KUKA KRL program: EPS_2_251806_MH04A_A_20260213065133.src

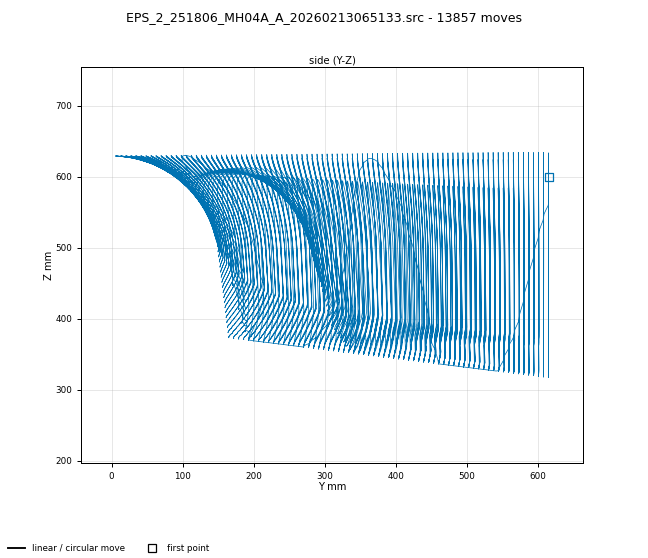
[picture p0: tool path of EPS_2_251806_MH04A_A_20260213065133.src, 13857 of 13859 moves have a stored position in this frame; points joined in program order, loops and branches not executed]
&ACCESS RVP
&REL 4
&COMMENT QRS 19112012
&PARAM EDITMASK = *
DEF PART()
EXT BAS (BAS_COMMAND :IN,REAL :IN )
INT I
BAS (#INITMOV,0 )

;KUKA QRS Post kuka4.cps  Date:22-06-2017 !

File_ID=3013

QRS_PRE_INIT()

;Init var - Until changes are made in qrs_pre_init
Outlet_Square_prg=0
Inlet_1_Square_prg=0
Inlet_2_Square_prg=0
Inlet_3_Square_prg=0
Inlet_4_Square_prg=0
Inlet_5_Square_prg=0

Outlet_1={X 0.000, Y 527.380, Z 509.000, B 0.000, E1 0.000 }
Inlet_1={X 0.000, Y 533.670, Z 484.000, B 0.000, E1 90.000 }
Inlet_2={X 0.000, Y 528.100, Z 499.000, B 0.000, E1 180.000 }
Outlet_1_type=251
Inlet_1_type=201
Inlet_2_type=251
;QRS#1=Sidecore dimensions
;QRS#2=250-10" PVC SDR 35
;QRS#3=200-8" PVC SDR 35
;QRS#4=250-10" PVC SDR 35
;QRS#5=
;QRS#6=
;QRS#7=
;QRS#8=
;QRS#9=14M PSX
;QRS#10=12-08 PSX
;QRS#11=14M PSX
;QRS#12=
;QRS#13=
;QRS#14=
;QRS#15=
;QRS#16=1220x127x914 3'
;QRS#17=EPS Height
;QRS#18=634,5
;QRS#19=*
;QRS#20= UPDATED VERSION 22-06-2017
;QRS#21=*
Outlet_Square=0100
Inlet_1_Square=0100
Inlet_2_Square=0100
Inlet_3_Square=0
Inlet_4_Square=0
Inlet_5_Square=0
Mill_Square=1
Outlet_Square_Prg=205
Inlet_1_Square_prg=204
Inlet_2_Square_prg=205

QRS_INIT()

$ADVANCE=5

; T1
PTP {E1 173.497,E2 173.497}
PTP {X 0,Y 615.499,A -85,B 0,C 180,E1 173.497,E2 173.497,E3 0,E4 0,E5 0,E6 0}
QRS_SPEED_INIT()
LIN {X 0,Y 615.499,Z 600,A -85,B 0,C 180,E1 173.497,E2 173.497,E3 0,E4 0,E5 0,E6 0} C_VEL
LIN {X 0,Y 615.499,Z 575.226,A -85,B 0,C 180,E1 173.497,E2 173.497} C_VEL
LIN {X 0,Y 615.499,Z 564.346,A -85,B 0,C 180,E1 173.497,E2 173.497} C_VEL
LIN {X 0,Y 615.497,Z 562.701,A -85,B 0,C 180,E1 173.417,E2 173.417} C_VEL
LIN {X 0,Y 615.497,Z 555.036,A -85,B 0,C 180,E1 172.455,E2 172.455} C_VEL
LIN {X 0,Y 615.498,Z 545.258,A -85,B 0,C 180,E1 171.463,E2 171.463} C_VEL
LIN {X 0,Y 615.497,Z 534.992,A -85,B 0,C 180,E1 170.636,E2 170.636} C_VEL
LIN {X 0,Y 615.479,Z 523.431,A -85,B 0,C 180,E1 169.888,E2 169.888} C_VEL
LIN {X 0,Y 615.498,Z 511.575,A -85,B 0,C 180,E1 169.293,E2 169.293} C_VEL
LIN {X 0,Y 615.483,Z 498.658,A -85,B 0,C 180,E1 168.807,E2 168.807} C_VEL
LIN {X 0,Y 615.49,Z 486.055,A -85,B 0,C 180,E1 168.473,E2 168.473} C_VEL
LIN {X 0,Y 615.489,Z 472.927,A -85,B 0,C 180,E1 168.264,E2 168.264} C_VEL
LIN {X 0,Y 615.486,Z 372.646,A -85,B 0,C 180,E1 167.072,E2 167.072} C_VEL
LIN {X 0,Y 615.491,Z 353.313,A -85,B 0,C 180,E1 164.265,E2 164.265} C_VEL
LIN {X 0,Y 615.488,Z 333.804,A -85,B 0,C 180,E1 161.396,E2 161.396} C_VEL
LIN {X 0,Y 615.479,Z 317.312,A -85,B 0,C 180,E1 158.919,E2 158.919} C_VEL
LIN {X 0,Y 615.487,Z 317.309,A -85,B 0,C 180,E1 156.444,E2 156.444} C_VEL
LIN {X 0,Y 615.483,Z 317.322,A -85,B 0,C 180,E1 153.556,E2 153.556} C_VEL
LIN {X 0,Y 615.471,Z 317.317,A -85,B 0,C 180,E1 151.341,E2 151.341} C_VEL
LIN {X 0,Y 615.479,Z 317.31,A -85,B 0,C 180,E1 148.916,E2 148.916} C_VEL
LIN {X 0,Y 615.496,Z 317.326,A -85,B 0,C 180,E1 145.978,E2 145.978} C_VEL
LIN {X 0,Y 615.464,Z 317.319,A -85,B 0,C 180,E1 143.573,E2 143.573} C_VEL
LIN {X 0,Y 615.474,Z 317.312,A -85,B 0,C 180,E1 140.94,E2 140.94} C_VEL
LIN {X 0,Y 615.471,Z 317.322,A -85,B 0,C 180,E1 137.922,E2 137.922} C_VEL
LIN {X 0,Y 615.46,Z 317.321,A -85,B 0,C 180,E1 135.848,E2 135.848} C_VEL
LIN {X 0,Y 615.467,Z 317.314,A -85,B 0,C 180,E1 133.045,E2 133.045} C_VEL
LIN {X 0,Y 615.461,Z 317.323,A -85,B 0,C 180,E1 130.086,E2 130.086} C_VEL
LIN {X 0,Y 615.449,Z 317.322,A -85,B 0,C 180,E1 128.007,E2 128.007} C_VEL
LIN {X 0,Y 615.432,Z 317.321,A -85,B 0,C 180,E1 125.62,E2 125.62} C_VEL
LIN {X 0,Y 615.447,Z 317.32,A -85,B 0,C 180,E1 123.239,E2 123.239} C_VEL
LIN {X 0,Y 615.486,Z 317.32,A -85,B 0,C 180,E1 120.921,E2 120.921} C_VEL
LIN {X 0,Y 615.457,Z 317.325,A -85,B 0,C 180,E1 118.445,E2 118.445} C_VEL
LIN {X 0,Y 615.45,Z 317.325,A -85,B 0,C 180,E1 116.447,E2 116.447} C_VEL
LIN {X 0,Y 615.412,Z 317.325,A -85,B 0,C 180,E1 113.992,E2 113.992} C_VEL
LIN {X 0,Y 615.422,Z 317.46,A -85,B 0,C 180,E1 111.633,E2 111.633} C_VEL
LIN {X 0,Y 615.493,Z 336.679,A -85,B 0,C 180,E1 108.992,E2 108.992} C_VEL
LIN {X 0,Y 615.483,Z 357.59,A -85,B 0,C 180,E1 106.166,E2 106.166} C_VEL
LIN {X 0,Y 615.491,Z 362.222,A -85,B 0,C 180,E1 105.545,E2 105.545} C_VEL
LIN {X 0,Y 615.497,Z 499.149,A -85,B 0,C 180,E1 103.905,E2 103.905} C_VEL
LIN {X 0,Y 615.493,Z 512.715,A -85,B 0,C 180,E1 103.622,E2 103.622} C_VEL
LIN {X 0,Y 615.495,Z 526.464,A -85,B 0,C 180,E1 103.202,E2 103.202} C_VEL
LIN {X 0,Y 615.495,Z 538.882,A -85,B 0,C 180,E1 102.698,E2 102.698} C_VEL
LIN {X 0,Y 615.495,Z 551.827,A -85,B 0,C 180,E1 102.029,E2 102.029} C_VEL
LIN {X 0,Y 615.499,Z 563.546,A -85,B 0,C 180,E1 101.277,E2 101.277} C_VEL
LIN {X 0,Y 615.498,Z 575.215,A -85,B 0,C 180,E1 100.361,E2 100.361} C_VEL
LIN {X 0,Y 615.497,Z 585.641,A -85,B 0,C 180,E1 99.365,E2 99.365} C_VEL
LIN {X 0,Y 615.496,Z 594.232,A -85,B 0,C 180,E1 98.372,E2 98.372} C_VEL
LIN {X 0,Y 615.495,Z 602.447,A -85,B 0,C 180,E1 97.216,E2 97.216} C_VEL
LIN {X 0,Y 615.496,Z 608.178,A -85,B 0,C 180,E1 96.228,E2 96.228} C_VEL
LIN {X 0,Y 615.491,Z 612.884,A -85,B 0,C 180,E1 95.242,E2 95.242} C_VEL
LIN {X 0,Y 615.496,Z 617.754,A -85,B 0,C 180,E1 93.929,E2 93.929} C_VEL
LIN {X 0,Y 615.496,Z 621.152,A -85,B 0,C 180,E1 92.619,E2 92.619} C_VEL
LIN {X 0,Y 615.493,Z 623.173,A -85,B 0,C 180,E1 91.31,E2 91.31} C_VEL
LIN {X 0,Y 615.494,Z 623.884,A -85,B 0,C 180,E1 90.001,E2 90.001} C_VEL
LIN {X 0,Y 615.49,Z 623.281,A -85,B 0,C 180,E1 88.692,E2 88.692} C_VEL
LIN {X 0,Y 615.493,Z 621.353,A -85,B 0,C 180,E1 87.383,E2 87.383} C_VEL
LIN {X 0,Y 615.496,Z 618.049,A -85,B 0,C 180,E1 86.073,E2 86.073} C_VEL
LIN {X 0,Y 615.496,Z 613.278,A -85,B 0,C 180,E1 84.76,E2 84.76} C_VEL
LIN {X 0,Y 615.494,Z 606.88,A -85,B 0,C 180,E1 83.444,E2 83.444} C_VEL
LIN {X 0,Y 615.496,Z 599.751,A -85,B 0,C 180,E1 82.291,E2 82.291} C_VEL
LIN {X 0,Y 615.497,Z 592.28,A -85,B 0,C 180,E1 81.299,E2 81.299} C_VEL
LIN {X 0,Y 615.495,Z 583.302,A -85,B 0,C 180,E1 80.305,E2 80.305} C_VEL
LIN {X 0,Y 615.499,Z 572.212,A -85,B 0,C 180,E1 79.291,E2 79.291} C_VEL
LIN {X 0,Y 615.498,Z 561.297,A -85,B 0,C 180,E1 78.475,E2 78.475} C_VEL
LIN {X 0,Y 615.488,Z 549.004,A -85,B 0,C 180,E1 77.722,E2 77.722} C_VEL
LIN {X 0,Y 615.498,Z 537.171,A -85,B 0,C 180,E1 77.136,E2 77.136} C_VEL
LIN {X 0,Y 615.492,Z 524.254,A -85,B 0,C 180,E1 76.632,E2 76.632} C_VEL
LIN {X 0,Y 615.495,Z 511.288,A -85,B 0,C 180,E1 76.253,E2 76.253} C_VEL
LIN {X 0,Y 615.493,Z 497.999,A -85,B 0,C 180,E1 75.988,E2 75.988} C_VEL
LIN {X 0,Y 615.493,Z 362.117,A -85,B 0,C 180,E1 74.351,E2 74.351} C_VEL
LIN {X 0,Y 615.477,Z 341.407,A -85,B 0,C 180,E1 71.559,E2 71.559} C_VEL
LIN {X 0,Y 615.491,Z 322.099,A -85,B 0,C 180,E1 68.921,E2 68.921} C_VEL
LIN {X 0,Y 615.426,Z 317.323,A -85,B 0,C 180,E1 68.237,E2 68.237} C_VEL
LIN {X 0,Y 615.432,Z 317.321,A -85,B 0,C 180,E1 65.727,E2 65.727} C_VEL
LIN {X 0,Y 615.473,Z 317.325,A -85,B 0,C 180,E1 62.824,E2 62.824} C_VEL
LIN {X 0,Y 615.42,Z 317.323,A -85,B 0,C 180,E1 60.217,E2 60.217} C_VEL
LIN {X 0,Y 615.425,Z 317.323,A -85,B 0,C 180,E1 58.313,E2 58.313} C_VEL
LIN {X 0,Y 615.422,Z 317.322,A -85,B 0,C 180,E1 55.976,E2 55.976} C_VEL
LIN {X 0,Y 615.449,Z 317.321,A -85,B 0,C 180,E1 53.574,E2 53.574} C_VEL
LIN {X 0,Y 615.478,Z 317.325,A -85,B 0,C 180,E1 50.939,E2 50.939} C_VEL
LIN {X 0,Y 615.432,Z 317.323,A -85,B 0,C 180,E1 48.523,E2 48.523} C_VEL
LIN {X 0,Y 615.422,Z 317.322,A -85,B 0,C 180,E1 46.009,E2 46.009} C_VEL
LIN {X 0,Y 615.499,Z 317.321,A -85,B 0,C 180,E1 43.244,E2 43.244} C_VEL
LIN {X 0,Y 615.433,Z 317.324,A -85,B 0,C 180,E1 40.611,E2 40.611} C_VEL
LIN {X 0,Y 615.462,Z 317.324,A -85,B 0,C 180,E1 38.906,E2 38.906} C_VEL
LIN {X 0,Y 615.422,Z 317.323,A -85,B 0,C 180,E1 36.429,E2 36.429} C_VEL
LIN {X 0,Y 615.467,Z 317.321,A -85,B 0,C 180,E1 33.534,E2 33.534} C_VEL
LIN {X 0,Y 615.456,Z 317.324,A -85,B 0,C 180,E1 30.922,E2 30.922} C_VEL
LIN {X 0,Y 615.419,Z 317.323,A -85,B 0,C 180,E1 28.442,E2 28.442} C_VEL
LIN {X 0,Y 615.419,Z 317.323,A -85,B 0,C 180,E1 26.447,E2 26.447} C_VEL
LIN {X 0,Y 615.426,Z 317.323,A -85,B 0,C 180,E1 23.999,E2 23.999} C_VEL
LIN {X 0,Y 615.489,Z 317.322,A -85,B 0,C 180,E1 21.432,E2 21.432} C_VEL
LIN {X 0,Y 615.421,Z 317.324,A -85,B 0,C 180,E1 18.591,E2 18.591} C_VEL
LIN {X 0,Y 615.415,Z 317.324,A -85,B 0,C 180,E1 16.414,E2 16.414} C_VEL
LIN {X 0,Y 615.435,Z 317.323,A -85,B 0,C 180,E1 13.92,E2 13.92} C_VEL
LIN {X 0,Y 615.433,Z 317.325,A -85,B 0,C 180,E1 10.87,E2 10.87} C_VEL
LIN {X 0,Y 615.416,Z 317.324,A -85,B 0,C 180,E1 8.538,E2 8.538} C_VEL
LIN {X 0,Y 615.413,Z 317.324,A -85,B 0,C 180,E1 6.533,E2 6.533} C_VEL
LIN {X 0,Y 615.415,Z 317.324,A -85,B 0,C 180,E1 4.585,E2 4.585} C_VEL
LIN {X 0,Y 615.417,Z 317.324,A -85,B 0,C 180,E1 2.618,E2 2.618} C_VEL
LIN {X 0,Y 615.417,Z 317.324,A -85,B 0,C 180,E1 0.654,E2 0.654} C_VEL
LIN {X 0,Y 615.418,Z 317.324,A -85,B 0,C 180,E1 -1.309,E2 -1.309} C_VEL
LIN {X 0,Y 615.419,Z 317.324,A -85,B 0,C 180,E1 -3.273,E2 -3.273} C_VEL
LIN {X 0,Y 615.419,Z 317.324,A -85,B 0,C 180,E1 -5.242,E2 -5.242} C_VEL
LIN {X 0,Y 615.417,Z 317.325,A -85,B 0,C 180,E1 -7.216,E2 -7.216} C_VEL
LIN {X 0,Y 615.419,Z 317.325,A -85,B 0,C 180,E1 -9.2,E2 -9.2} C_VEL
LIN {X 0,Y 615.419,Z 317.324,A -85,B 0,C 180,E1 -11.194,E2 -11.194} C_VEL
LIN {X 0,Y 615.418,Z 317.324,A -85,B 0,C 180,E1 -13.203,E2 -13.203} C_VEL
LIN {X 0,Y 615.416,Z 317.324,A -85,B 0,C 180,E1 -15.228,E2 -15.228} C_VEL
LIN {X 0,Y 615.414,Z 317.324,A -85,B 0,C 180,E1 -17.273,E2 -17.273} C_VEL
LIN {X 0,Y 615.412,Z 317.324,A -85,B 0,C 180,E1 -19.34,E2 -19.34} C_VEL
LIN {X 0,Y 615.411,Z 317.324,A -85,B 0,C 180,E1 -21.435,E2 -21.435} C_VEL
LIN {X 0,Y 615.411,Z 317.325,A -85,B 0,C 180,E1 -23.559,E2 -23.559} C_VEL
LIN {X 0,Y 615.489,Z 317.325,A -85,B 0,C 180,E1 -26.444,E2 -26.444} C_VEL
LIN {X 0,Y 615.455,Z 317.325,A -85,B 0,C 180,E1 -28.66,E2 -28.66} C_VEL
LIN {X 0,Y 615.416,Z 317.325,A -85,B 0,C 180,E1 -31.078,E2 -31.078} C_VEL
LIN {X 0,Y 615.41,Z 317.325,A -85,B 0,C 180,E1 -33.241,E2 -33.241} C_VEL
LIN {X 0,Y 615.435,Z 317.325,A -85,B 0,C 180,E1 -35.83,E2 -35.83} C_VEL
LIN {X 0,Y 615.465,Z 317.325,A -85,B 0,C 180,E1 -38.07,E2 -38.07} C_VEL
LIN {X 0,Y 615.45,Z 317.325,A -85,B 0,C 180,E1 -40.609,E2 -40.609} C_VEL
LIN {X 0,Y 615.413,Z 317.325,A -85,B 0,C 180,E1 -43.042,E2 -43.042} C_VEL
LIN {X 0,Y 615.411,Z 317.325,A -85,B 0,C 180,E1 -45.076,E2 -45.076} C_VEL
LIN {X 0,Y 615.424,Z 317.325,A -85,B 0,C 180,E1 -47.644,E2 -47.644} C_VEL
LIN {X 0,Y 615.488,Z 317.326,A -85,B 0,C 180,E1 -50.252,E2 -50.252} C_VEL
LIN {X 0,Y 615.427,Z 317.325,A -85,B 0,C 180,E1 -52.755,E2 -52.755} C_VEL
LIN {X 0,Y 615.41,Z 317.325,A -85,B 0,C 180,E1 -55.182,E2 -55.182} C_VEL
LIN {X 0,Y 615.433,Z 317.325,A -85,B 0,C 180,E1 -57.678,E2 -57.678} C_VEL
LIN {X 0,Y 615.439,Z 317.324,A -85,B 0,C 180,E1 -60.593,E2 -60.593} C_VEL
LIN {X 0,Y 615.413,Z 317.324,A -85,B 0,C 180,E1 -62.969,E2 -62.969} C_VEL
LIN {X 0,Y 615.412,Z 317.324,A -85,B 0,C 180,E1 -65.006,E2 -65.006} C_VEL
LIN {X 0,Y 615.418,Z 317.458,A -85,B 0,C 180,E1 -67.378,E2 -67.378} C_VEL
LIN {X 0,Y 615.484,Z 337.246,A -85,B 0,C 180,E1 -69.968,E2 -69.968} C_VEL
LIN {X 0,Y 615.486,Z 358.699,A -85,B 0,C 180,E1 -72.731,E2 -72.731} C_VEL
LIN {X 0,Y 615.493,Z 372.139,A -85,B 0,C 180,E1 -74.415,E2 -74.415} C_VEL
LIN {X 0,Y 615.499,Z 509.922,A -85,B 0,C 180,E1 -76.064,E2 -76.064} C_VEL
LIN {X 0,Y 615.495,Z 524.419,A -85,B 0,C 180,E1 -76.38,E2 -76.38} C_VEL
LIN {X 0,Y 615.489,Z 537.719,A -85,B 0,C 180,E1 -76.8,E2 -76.8} C_VEL
LIN {X 0,Y 615.498,Z 551.606,A -85,B 0,C 180,E1 -77.387,E2 -77.387} C_VEL
LIN {X 0,Y 615.495,Z 564.026,A -85,B 0,C 180,E1 -78.057,E2 -78.057} C_VEL
LIN {X 0,Y 615.499,Z 575.356,A -85,B 0,C 180,E1 -78.808,E2 -78.808} C_VEL
LIN {X 0,Y 615.498,Z 585.761,A -85,B 0,C 180,E1 -79.641,E2 -79.641} C_VEL
LIN {X 0,Y 615.496,Z 596.099,A -85,B 0,C 180,E1 -80.637,E2 -80.637} C_VEL
LIN {X 0,Y 615.497,Z 604.611,A -85,B 0,C 180,E1 -81.63,E2 -81.63} C_VEL
LIN {X 0,Y 615.496,Z 612.733,A -85,B 0,C 180,E1 -82.786,E2 -82.786} C_VEL
LIN {X 0,Y 615.496,Z 618.436,A -85,B 0,C 180,E1 -83.774,E2 -83.774} C_VEL
LIN {X 0,Y 615.495,Z 623.085,A -85,B 0,C 180,E1 -84.76,E2 -84.76} C_VEL
LIN {X 0,Y 615.494,Z 627.905,A -85,B 0,C 180,E1 -86.073,E2 -86.073} C_VEL
LIN {X 0,Y 615.496,Z 631.254,A -85,B 0,C 180,E1 -87.383,E2 -87.383} C_VEL
LIN {X 0,Y 615.489,Z 633.23,A -85,B 0,C 180,E1 -88.692,E2 -88.692} C_VEL
LIN {X 0,Y 615.493,Z 633.889,A -85,B 0,C 180,E1 -90.001,E2 -90.001} C_VEL
LIN {X 0,Y 615.489,Z 633.227,A -85,B 0,C 180,E1 -91.31,E2 -91.31} C_VEL
LIN {X 0,Y 615.496,Z 631.25,A -85,B 0,C 180,E1 -92.619,E2 -92.619} C_VEL
LIN {X 0,Y 615.494,Z 627.898,A -85,B 0,C 180,E1 -93.929,E2 -93.929} C_VEL
LIN {X 0,Y 615.495,Z 623.076,A -85,B 0,C 180,E1 -95.242,E2 -95.242} C_VEL
LIN {X 0,Y 615.496,Z 616.623,A -85,B 0,C 180,E1 -96.557,E2 -96.557} C_VEL
LIN {X 0,Y 615.497,Z 609.434,A -85,B 0,C 180,E1 -97.711,E2 -97.711} C_VEL
LIN {X 0,Y 615.497,Z 601.896,A -85,B 0,C 180,E1 -98.703,E2 -98.703} C_VEL
LIN {X 0,Y 615.495,Z 592.844,A -85,B 0,C 180,E1 -99.697,E2 -99.697} C_VEL
LIN {X 0,Y 615.497,Z 582.75,A -85,B 0,C 180,E1 -100.619,E2 -100.619} C_VEL
LIN {X 0,Y 615.498,Z 571.844,A -85,B 0,C 180,E1 -101.444,E2 -101.444} C_VEL
LIN {X 0,Y 615.489,Z 559.689,A -85,B 0,C 180,E1 -102.196,E2 -102.196} C_VEL
LIN {X 0,Y 615.498,Z 546.069,A -85,B 0,C 180,E1 -102.866,E2 -102.866} C_VEL
LIN {X 0,Y 615.49,Z 532.807,A -85,B 0,C 180,E1 -103.37,E2 -103.37} C_VEL
LIN {X 0,Y 615.494,Z 519.247,A -85,B 0,C 180,E1 -103.749,E2 -103.749} C_VEL
LIN {X 0,Y 615.496,Z 504.72,A -85,B 0,C 180,E1 -104.013,E2 -104.013} C_VEL
LIN {X 0,Y 615.494,Z 371.744,A -85,B 0,C 180,E1 -105.608,E2 -105.608} C_VEL
LIN {X 0,Y 615.482,Z 349.549,A -85,B 0,C 180,E1 -108.442,E2 -108.442} C_VEL
LIN {X 0,Y 615.485,Z 329.177,A -85,B 0,C 180,E1 -111.082,E2 -111.082} C_VEL
LIN {X 0,Y 615.419,Z 317.325,A -85,B 0,C 180,E1 -112.656,E2 -112.656} C_VEL
LIN {X 0,Y 615.423,Z 317.324,A -85,B 0,C 180,E1 -114.995,E2 -114.995} C_VEL
LIN {X 0,Y 615.443,Z 317.324,A -85,B 0,C 180,E1 -117.18,E2 -117.18} C_VEL
LIN {X 0,Y 615.457,Z 317.318,A -85,B 0,C 180,E1 -120.162,E2 -120.162} C_VEL
LIN {X 0,Y 615.446,Z 317.318,A -85,B 0,C 180,E1 -122.461,E2 -122.461} C_VEL
LIN {X 0,Y 615.456,Z 317.321,A -85,B 0,C 180,E1 -124.818,E2 -124.818} C_VEL
LIN {X 0,Y 615.492,Z 317.325,A -85,B 0,C 180,E1 -127.243,E2 -127.243} C_VEL
LIN {X 0,Y 615.473,Z 317.312,A -85,B 0,C 180,E1 -130.087,E2 -130.087} C_VEL
LIN {X 0,Y 615.468,Z 317.316,A -85,B 0,C 180,E1 -132.355,E2 -132.355} C_VEL
LIN {X 0,Y 615.486,Z 317.32,A -85,B 0,C 180,E1 -135.069,E2 -135.069} C_VEL
LIN {X 0,Y 615.487,Z 317.31,A -85,B 0,C 180,E1 -137.921,E2 -137.921} C_VEL
LIN {X 0,Y 615.484,Z 317.318,A -85,B 0,C 180,E1 -140.25,E2 -140.25} C_VEL
LIN {X 0,Y 615.464,Z 317.317,A -85,B 0,C 180,E1 -143.067,E2 -143.067} C_VEL
LIN {X 0,Y 615.467,Z 317.313,A -85,B 0,C 180,E1 -145.303,E2 -145.303} C_VEL
LIN {X 0,Y 615.494,Z 317.311,A -85,B 0,C 180,E1 -147.669,E2 -147.669} C_VEL
LIN {X 0,Y 615.454,Z 317.321,A -85,B 0,C 180,E1 -150.592,E2 -150.592} C_VEL
LIN {X 0,Y 615.441,Z 317.319,A -85,B 0,C 180,E1 -152.964,E2 -152.964} C_VEL
LIN {X 0,Y 615.495,Z 317.321,A -85,B 0,C 180,E1 -155.728,E2 -155.728} C_VEL
LIN {X 0,Y 615.479,Z 317.326,A -85,B 0,C 180,E1 -157.863,E2 -157.863} C_VEL
LIN {X 0,Y 615.433,Z 317.48,A -85,B 0,C 180,E1 -159.049,E2 -159.049} C_VEL
LIN {X 0,Y 615.496,Z 335.382,A -85,B 0,C 180,E1 -161.72,E2 -161.72} C_VEL
LIN {X 0,Y 615.498,Z 355.023,A -85,B 0,C 180,E1 -164.605,E2 -164.605} C_VEL
LIN {X 0,Y 615.49,Z 372.749,A -85,B 0,C 180,E1 -167.177,E2 -167.177} C_VEL
LIN {X 0,Y 615.493,Z 480.144,A -85,B 0,C 180,E1 -168.453,E2 -168.453} C_VEL
LIN {X 0,Y 615.491,Z 492.724,A -85,B 0,C 180,E1 -168.724,E2 -168.724} C_VEL
LIN {X 0,Y 615.491,Z 506.106,A -85,B 0,C 180,E1 -169.158,E2 -169.158} C_VEL
LIN {X 0,Y 615.492,Z 517.066,A -85,B 0,C 180,E1 -169.639,E2 -169.639} C_VEL
LIN {X 0,Y 615.482,Z 528.806,A -85,B 0,C 180,E1 -170.304,E2 -170.304} C_VEL
LIN {X 0,Y 615.499,Z 539.268,A -85,B 0,C 180,E1 -171.05,E2 -171.05} C_VEL
LIN {X 0,Y 615.498,Z 547.831,A -85,B 0,C 180,E1 -171.794,E2 -171.794} C_VEL
LIN {X 0,Y 615.498,Z 555.709,A -85,B 0,C 180,E1 -172.62,E2 -172.62} C_VEL
LIN {X 0,Y 615.497,Z 563.399,A -85,B 0,C 180,E1 -173.608,E2 -173.608} C_VEL
LIN {X 0,Y 615.498,Z 570.458,A -85,B 0,C 180,E1 -174.759,E2 -174.759} C_VEL
LIN {X 0,Y 615.493,Z 575.158,A -85,B 0,C 180,E1 -175.744,E2 -175.744} C_VEL
LIN {X 0,Y 615.496,Z 578.754,A -85,B 0,C 180,E1 -176.727,E2 -176.727} C_VEL
LIN {X 0,Y 615.496,Z 580.615,A -85,B 0,C 180,E1 -177.382,E2 -177.382} C_VEL
LIN {X 0,Y 615.497,Z 582.034,A -85,B 0,C 180,E1 -178.037,E2 -178.037} C_VEL
LIN {X 0,Y 615.496,Z 583.642,A -85,B 0,C 180,E1 -179.346,E2 -179.346} C_VEL
LIN {X 0,Y 615.494,Z 583.884,A -85,B 0,C 180,E1 -180,E2 -180} C_VEL
LIN {X 0,Y 615.496,Z 583.705,A -85,B 0,C 180,E1 -180.654,E2 -180.654} C_VEL
LIN {X 0,Y 615.496,Z 582.183,A -85,B 0,C 180,E1 -181.963,E2 -181.963} C_VEL
LIN {X 0,Y 615.498,Z 580.841,A -85,B 0,C 180,E1 -182.618,E2 -182.618} C_VEL
LIN {X 0,Y 615.497,Z 577.994,A -85,B 0,C 180,E1 -183.601,E2 -183.601} C_VEL
LIN {X 0,Y 615.499,Z 574.134,A -85,B 0,C 180,E1 -184.585,E2 -184.585} C_VEL
LIN {X 0,Y 615.498,Z 569.151,A -85,B 0,C 180,E1 -185.57,E2 -185.57} C_VEL
LIN {X 0,Y 615.497,Z 562.701,A -85,B 0,C 180,E1 -186.583,E2 -186.583} C_VEL
LIN {X 0,Y 614.829,Z 559.52,A -85,B 0,C 180,E1 -187.032,E2 -187.032} C_VEL
LIN {X 0,Y 611.988,Z 553.946,A -85,B 0,C 180,E1 -187.749,E2 -187.749} C_VEL
LIN {X 0,Y 609.138,Z 547.67,A -85,B 0,C 180,E1 -188.43,E2 -188.43} C_VEL
LIN {X 0,Y 608.477,Z 543.429,A -85,B 0,C 180,E1 -188.82,E2 -188.82} C_VEL
LIN {X 0,Y 608.489,Z 532.886,A -85,B 0,C 180,E1 -189.641,E2 -189.641} C_VEL
LIN {X 0,Y 608.49,Z 522.11,A -85,B 0,C 180,E1 -190.313,E2 -190.313} C_VEL
LIN {X 0,Y 608.52,Z 509.659,A -85,B 0,C 180,E1 -190.919,E2 -190.919} C_VEL
LIN {X 0,Y 608.522,Z 497.464,A -85,B 0,C 180,E1 -191.365,E2 -191.365} C_VEL
LIN {X 0,Y 608.549,Z 485.156,A -85,B 0,C 180,E1 -191.681,E2 -191.681} C_VEL
LIN {X 0,Y 608.556,Z 471.245,A -85,B 0,C 180,E1 -191.892,E2 -191.892} C_VEL
LIN {X 0,Y 608.466,Z 372.952,A -85,B 0,C 180,E1 -193.059,E2 -193.059} C_VEL
LIN {X 0,Y 608.492,Z 353.399,A -85,B 0,C 180,E1 -195.921,E2 -195.921} C_VEL
LIN {X 0,Y 608.515,Z 334.494,A -85,B 0,C 180,E1 -198.727,E2 -198.727} C_VEL
LIN {X 0,Y 608.476,Z 318.312,A -85,B 0,C 180,E1 -201.18,E2 -201.18} C_VEL
LIN {X 0,Y 608.465,Z 318.314,A -85,B 0,C 180,E1 -203.845,E2 -203.845} C_VEL
LIN {X 0,Y 608.443,Z 318.321,A -85,B 0,C 180,E1 -206.036,E2 -206.036} C_VEL
LIN {X 0,Y 608.464,Z 318.315,A -85,B 0,C 180,E1 -208.618,E2 -208.618} C_VEL
LIN {X 0,Y 608.449,Z 318.314,A -85,B 0,C 180,E1 -211.318,E2 -211.318} C_VEL
LIN {X 0,Y 608.477,Z 318.315,A -85,B 0,C 180,E1 -213.735,E2 -213.735} C_VEL
LIN {X 0,Y 608.447,Z 318.322,A -85,B 0,C 180,E1 -216.092,E2 -216.092} C_VEL
LIN {X 0,Y 608.427,Z 318.317,A -85,B 0,C 180,E1 -218.591,E2 -218.591} C_VEL
LIN {X 0,Y 608.462,Z 318.314,A -85,B 0,C 180,E1 -221.341,E2 -221.341} C_VEL
LIN {X 0,Y 608.462,Z 318.32,A -85,B 0,C 180,E1 -223.87,E2 -223.87} C_VEL
LIN {X 0,Y 608.445,Z 318.314,A -85,B 0,C 180,E1 -226.694,E2 -226.694} C_VEL
LIN {X 0,Y 608.427,Z 318.316,A -85,B 0,C 180,E1 -228.82,E2 -228.82} C_VEL
LIN {X 0,Y 608.445,Z 318.32,A -85,B 0,C 180,E1 -231.763,E2 -231.763} C_VEL
LIN {X 0,Y 608.434,Z 318.318,A -85,B 0,C 180,E1 -233.957,E2 -233.957} C_VEL
LIN {X 0,Y 608.415,Z 318.317,A -85,B 0,C 180,E1 -236.325,E2 -236.325} C_VEL
LIN {X 0,Y 608.438,Z 318.316,A -85,B 0,C 180,E1 -238.734,E2 -238.734} C_VEL
LIN {X 0,Y 608.41,Z 318.321,A -85,B 0,C 180,E1 -241.73,E2 -241.73} C_VEL
LIN {X 0,Y 608.394,Z 318.32,A -85,B 0,C 180,E1 -244.295,E2 -244.295} C_VEL
LIN {X 0,Y 608.421,Z 318.323,A -85,B 0,C 180,E1 -246.874,E2 -246.874} C_VEL
LIN {X 0,Y 608.402,Z 318.419,A -85,B 0,C 180,E1 -248.238,E2 -248.238} C_VEL
LIN {X 0,Y 608.546,Z 332.889,A -85,B 0,C 180,E1 -250.256,E2 -250.256} C_VEL
LIN {X 0,Y 608.505,Z 353.244,A -85,B 0,C 180,E1 -253.044,E2 -253.044} C_VEL
LIN {X 0,Y 608.512,Z 362.308,A -85,B 0,C 180,E1 -254.272,E2 -254.272} C_VEL
LIN {X 0,Y 608.614,Z 474.489,A -85,B 0,C 180,E1 -255.624,E2 -255.624} C_VEL
LIN {X 0,Y 608.611,Z 500.869,A -85,B 0,C 180,E1 -255.965,E2 -255.965} C_VEL
LIN {X 0,Y 608.6,Z 515.036,A -85,B 0,C 180,E1 -256.284,E2 -256.284} C_VEL
LIN {X 0,Y 608.576,Z 528.741,A -85,B 0,C 180,E1 -256.73,E2 -256.73} C_VEL
LIN {X 0,Y 608.545,Z 540.673,A -85,B 0,C 180,E1 -257.239,E2 -257.239} C_VEL
LIN {X 0,Y 608.534,Z 553.325,A -85,B 0,C 180,E1 -257.916,E2 -257.916} C_VEL
LIN {X 0,Y 608.5,Z 564.841,A -85,B 0,C 180,E1 -258.676,E2 -258.676} C_VEL
LIN {X 0,Y 608.495,Z 575.404,A -85,B 0,C 180,E1 -259.518,E2 -259.518} C_VEL
LIN {X 0,Y 608.48,Z 585.89,A -85,B 0,C 180,E1 -260.526,E2 -260.526} C_VEL
LIN {X 0,Y 608.463,Z 594.542,A -85,B 0,C 180,E1 -261.53,E2 -261.53} C_VEL
LIN {X 0,Y 608.461,Z 602.833,A -85,B 0,C 180,E1 -262.7,E2 -262.7} C_VEL
LIN {X 0,Y 608.443,Z 609.322,A -85,B 0,C 180,E1 -263.831,E2 -263.831} C_VEL
LIN {X 0,Y 608.437,Z 614.784,A -85,B 0,C 180,E1 -265.029,E2 -265.029} C_VEL
LIN {X 0,Y 608.434,Z 618.295,A -85,B 0,C 180,E1 -266.025,E2 -266.025} C_VEL
LIN {X 0,Y 608.424,Z 621.731,A -85,B 0,C 180,E1 -267.351,E2 -267.351} C_VEL
LIN {X 0,Y 608.446,Z 623.775,A -85,B 0,C 180,E1 -268.675,E2 -268.675} C_VEL
LIN {X 0,Y 608.434,Z 624.495,A -85,B 0,C 180,E1 -269.999,E2 -269.999} C_VEL
LIN {X 0,Y 608.443,Z 623.883,A -85,B 0,C 180,E1 -271.323,E2 -271.323} C_VEL
LIN {X 0,Y 608.421,Z 621.93,A -85,B 0,C 180,E1 -272.647,E2 -272.647} C_VEL
LIN {X 0,Y 608.434,Z 618.589,A -85,B 0,C 180,E1 -273.973,E2 -273.973} C_VEL
LIN {X 0,Y 608.44,Z 613.765,A -85,B 0,C 180,E1 -275.301,E2 -275.301} C_VEL
LIN {X 0,Y 608.438,Z 607.302,A -85,B 0,C 180,E1 -276.632,E2 -276.632} C_VEL
LIN {X 0,Y 608.453,Z 600.105,A -85,B 0,C 180,E1 -277.799,E2 -277.799} C_VEL
LIN {X 0,Y 608.476,Z 592.57,A -85,B 0,C 180,E1 -278.802,E2 -278.802} C_VEL
LIN {X 0,Y 608.486,Z 583.53,A -85,B 0,C 180,E1 -279.808,E2 -279.808} C_VEL
LIN {X 0,Y 608.507,Z 572.723,A -85,B 0,C 180,E1 -280.804,E2 -280.804} C_VEL
LIN {X 0,Y 608.523,Z 561.397,A -85,B 0,C 180,E1 -281.659,E2 -281.659} C_VEL
LIN {X 0,Y 608.539,Z 549.064,A -85,B 0,C 180,E1 -282.42,E2 -282.42} C_VEL
LIN {X 0,Y 608.56,Z 537.201,A -85,B 0,C 180,E1 -283.013,E2 -283.013} C_VEL
LIN {X 0,Y 608.58,Z 524.252,A -85,B 0,C 180,E1 -283.523,E2 -283.523} C_VEL
LIN {X 0,Y 608.592,Z 510.002,A -85,B 0,C 180,E1 -283.935,E2 -283.935} C_VEL
LIN {X 0,Y 608.607,Z 496.676,A -85,B 0,C 180,E1 -284.192,E2 -284.192} C_VEL
LIN {X 0,Y 608.514,Z 362.354,A -85,B 0,C 180,E1 -285.812,E2 -285.812} C_VEL
LIN {X 0,Y 608.504,Z 342.624,A -85,B 0,C 180,E1 -288.496,E2 -288.496} C_VEL
LIN {X 0,Y 608.557,Z 323.373,A -85,B 0,C 180,E1 -291.154,E2 -291.154} C_VEL
LIN {X 0,Y 608.415,Z 318.319,A -85,B 0,C 180,E1 -291.87,E2 -291.87} C_VEL
LIN {X 0,Y 608.43,Z 318.319,A -85,B 0,C 180,E1 -294.571,E2 -294.571} C_VEL
LIN {X 0,Y 608.417,Z 318.319,A -85,B 0,C 180,E1 -297.518,E2 -297.518} C_VEL
LIN {X 0,Y 608.392,Z 318.32,A -85,B 0,C 180,E1 -299.959,E2 -299.959} C_VEL
LIN {X 0,Y 608.431,Z 318.318,A -85,B 0,C 180,E1 -302.517,E2 -302.517} C_VEL
LIN {X 0,Y 608.415,Z 318.322,A -85,B 0,C 180,E1 -305.278,E2 -305.278} C_VEL
LIN {X 0,Y 608.4,Z 318.319,A -85,B 0,C 180,E1 -307.75,E2 -307.75} C_VEL
LIN {X 0,Y 608.424,Z 318.318,A -85,B 0,C 180,E1 -310.326,E2 -310.326} C_VEL
LIN {X 0,Y 608.44,Z 318.318,A -85,B 0,C 180,E1 -313.306,E2 -313.306} C_VEL
LIN {X 0,Y 608.419,Z 318.317,A -85,B 0,C 180,E1 -316.126,E2 -316.126} C_VEL
LIN {X 0,Y 608.445,Z 318.324,A -85,B 0,C 180,E1 -318.822,E2 -318.822} C_VEL
LIN {X 0,Y 608.402,Z 318.32,A -85,B 0,C 180,E1 -321.407,E2 -321.407} C_VEL
LIN {X 0,Y 608.432,Z 318.321,A -85,B 0,C 180,E1 -323.083,E2 -323.083} C_VEL
LIN {X 0,Y 608.42,Z 318.317,A -85,B 0,C 180,E1 -325.527,E2 -325.527} C_VEL
LIN {X 0,Y 608.413,Z 318.317,A -85,B 0,C 180,E1 -327.902,E2 -327.902} C_VEL
LIN {X 0,Y 608.426,Z 318.318,A -85,B 0,C 180,E1 -330.218,E2 -330.218} C_VEL
LIN {X 0,Y 608.409,Z 318.32,A -85,B 0,C 180,E1 -333.224,E2 -333.224} C_VEL
LIN {X 0,Y 608.399,Z 318.319,A -85,B 0,C 180,E1 -335.86,E2 -335.86} C_VEL
LIN {X 0,Y 608.445,Z 318.317,A -85,B 0,C 180,E1 -338.307,E2 -338.307} C_VEL
LIN {X 0,Y 608.405,Z 318.32,A -85,B 0,C 180,E1 -341.297,E2 -341.297} C_VEL
LIN {X 0,Y 608.404,Z 318.319,A -85,B 0,C 180,E1 -343.905,E2 -343.905} C_VEL
LIN {X 0,Y 608.445,Z 318.324,A -85,B 0,C 180,E1 -346.643,E2 -346.643} C_VEL
LIN {X 0,Y 608.402,Z 318.319,A -85,B 0,C 180,E1 -349.349,E2 -349.349} C_VEL
LIN {X 0,Y 608.4,Z 318.319,A -85,B 0,C 180,E1 -351.363,E2 -351.363} C_VEL
LIN {X 0,Y 608.396,Z 318.32,A -85,B 0,C 180,E1 -353.421,E2 -353.421} C_VEL
LIN {X 0,Y 608.389,Z 318.321,A -85,B 0,C 180,E1 -355.362,E2 -355.362} C_VEL
LIN {X 0,Y 608.415,Z 318.317,A -85,B 0,C 180,E1 -357.352,E2 -357.352} C_VEL
LIN {X 0,Y 608.396,Z 318.32,A -85,B 0,C 180,E1 -359.338,E2 -359.338} C_VEL
LIN {X 0,Y 608.407,Z 318.318,A -85,B 0,C 180,E1 -361.324,E2 -361.324} C_VEL
LIN {X 0,Y 608.388,Z 318.321,A -85,B 0,C 180,E1 -363.311,E2 -363.311} C_VEL
LIN {X 0,Y 608.402,Z 318.319,A -85,B 0,C 180,E1 -365.302,E2 -365.302} C_VEL
LIN {X 0,Y 608.394,Z 318.32,A -85,B 0,C 180,E1 -367.3,E2 -367.3} C_VEL
LIN {X 0,Y 608.407,Z 318.318,A -85,B 0,C 180,E1 -369.307,E2 -369.307} C_VEL
LIN {X 0,Y 608.396,Z 318.319,A -85,B 0,C 180,E1 -371.325,E2 -371.325} C_VEL
LIN {X 0,Y 608.401,Z 318.319,A -85,B 0,C 180,E1 -373.358,E2 -373.358} C_VEL
LIN {X 0,Y 608.41,Z 318.318,A -85,B 0,C 180,E1 -375.408,E2 -375.408} C_VEL
LIN {X 0,Y 608.393,Z 318.32,A -85,B 0,C 180,E1 -377.478,E2 -377.478} C_VEL
LIN {X 0,Y 608.395,Z 318.32,A -85,B 0,C 180,E1 -379.572,E2 -379.572} C_VEL
LIN {X 0,Y 608.416,Z 318.317,A -85,B 0,C 180,E1 -381.694,E2 -381.694} C_VEL
LIN {X 0,Y 608.425,Z 318.323,A -85,B 0,C 180,E1 -384.572,E2 -384.572} C_VEL
LIN {X 0,Y 608.398,Z 318.319,A -85,B 0,C 180,E1 -387.196,E2 -387.196} C_VEL
LIN {X 0,Y 608.391,Z 318.321,A -85,B 0,C 180,E1 -389.024,E2 -389.024} C_VEL
LIN {X 0,Y 608.392,Z 318.32,A -85,B 0,C 180,E1 -391.321,E2 -391.321} C_VEL
LIN {X 0,Y 608.41,Z 318.319,A -85,B 0,C 180,E1 -393.729,E2 -393.729} C_VEL
LIN {X 0,Y 608.426,Z 318.322,A -85,B 0,C 180,E1 -396.094,E2 -396.094} C_VEL
LIN {X 0,Y 608.394,Z 318.325,A -85,B 0,C 180,E1 -398.594,E2 -398.594} C_VEL
LIN {X 0,Y 608.381,Z 318.321,A -85,B 0,C 180,E1 -401.183,E2 -401.183} C_VEL
LIN {X 0,Y 608.405,Z 318.318,A -85,B 0,C 180,E1 -403.304,E2 -403.304} C_VEL
LIN {X 0,Y 608.444,Z 318.322,A -85,B 0,C 180,E1 -406.13,E2 -406.13} C_VEL
LIN {X 0,Y 608.395,Z 318.321,A -85,B 0,C 180,E1 -408.82,E2 -408.82} C_VEL
LIN {X 0,Y 608.383,Z 318.321,A -85,B 0,C 180,E1 -411.407,E2 -411.407} C_VEL
LIN {X 0,Y 608.433,Z 318.321,A -85,B 0,C 180,E1 -413.956,E2 -413.956} C_VEL
LIN {X 0,Y 608.435,Z 318.322,A -85,B 0,C 180,E1 -416.329,E2 -416.329} C_VEL
LIN {X 0,Y 608.419,Z 318.318,A -85,B 0,C 180,E1 -418.737,E2 -418.737} C_VEL
LIN {X 0,Y 608.387,Z 318.321,A -85,B 0,C 180,E1 -420.977,E2 -420.977} C_VEL
LIN {X 0,Y 608.383,Z 318.321,A -85,B 0,C 180,E1 -423.224,E2 -423.224} C_VEL
LIN {X 0,Y 608.406,Z 318.319,A -85,B 0,C 180,E1 -425.428,E2 -425.428} C_VEL
LIN {X 0,Y 608.404,Z 318.455,A -85,B 0,C 180,E1 -427.235,E2 -427.235} C_VEL
LIN {X 0,Y 608.582,Z 331.88,A -85,B 0,C 180,E1 -429.024,E2 -429.024} C_VEL
LIN {X 0,Y 608.531,Z 353.364,A -85,B 0,C 180,E1 -431.832,E2 -431.832} C_VEL
LIN {X 0,Y 608.547,Z 372.139,A -85,B 0,C 180,E1 -434.232,E2 -434.232} C_VEL
LIN {X 0,Y 608.618,Z 508.983,A -85,B 0,C 180,E1 -435.886,E2 -435.886} C_VEL
LIN {X 0,Y 608.594,Z 523.665,A -85,B 0,C 180,E1 -436.201,E2 -436.201} C_VEL
LIN {X 0,Y 608.579,Z 537.74,A -85,B 0,C 180,E1 -436.647,E2 -436.647} C_VEL
LIN {X 0,Y 608.565,Z 549.907,A -85,B 0,C 180,E1 -437.157,E2 -437.157} C_VEL
LIN {X 0,Y 608.516,Z 562.7,A -85,B 0,C 180,E1 -437.833,E2 -437.833} C_VEL
LIN {X 0,Y 608.499,Z 575.486,A -85,B 0,C 180,E1 -438.678,E2 -438.678} C_VEL
LIN {X 0,Y 608.495,Z 585.944,A -85,B 0,C 180,E1 -439.52,E2 -439.52} C_VEL
LIN {X 0,Y 608.479,Z 596.345,A -85,B 0,C 180,E1 -440.528,E2 -440.528} C_VEL
LIN {X 0,Y 608.464,Z 604.922,A -85,B 0,C 180,E1 -441.532,E2 -441.532} C_VEL
LIN {X 0,Y 608.461,Z 613.12,A -85,B 0,C 180,E1 -442.702,E2 -442.702} C_VEL
LIN {X 0,Y 608.443,Z 619.548,A -85,B 0,C 180,E1 -443.831,E2 -443.831} C_VEL
LIN {X 0,Y 608.438,Z 624.966,A -85,B 0,C 180,E1 -445.031,E2 -445.031} C_VEL
LIN {X 0,Y 608.431,Z 628.445,A -85,B 0,C 180,E1 -446.027,E2 -446.027} C_VEL
LIN {X 0,Y 608.424,Z 631.833,A -85,B 0,C 180,E1 -447.353,E2 -447.353} C_VEL
LIN {X 0,Y 608.442,Z 633.832,A -85,B 0,C 180,E1 -448.677,E2 -448.677} C_VEL
LIN {X 0,Y 608.433,Z 634.5,A -85,B 0,C 180,E1 -450.001,E2 -450.001} C_VEL
LIN {X 0,Y 608.442,Z 633.829,A -85,B 0,C 180,E1 -451.325,E2 -451.325} C_VEL
LIN {X 0,Y 608.424,Z 631.829,A -85,B 0,C 180,E1 -452.649,E2 -452.649} C_VEL
LIN {X 0,Y 608.431,Z 628.438,A -85,B 0,C 180,E1 -453.975,E2 -453.975} C_VEL
LIN {X 0,Y 608.44,Z 623.563,A -85,B 0,C 180,E1 -455.303,E2 -455.303} C_VEL
LIN {X 0,Y 608.446,Z 617.207,A -85,B 0,C 180,E1 -456.604,E2 -456.604} C_VEL
LIN {X 0,Y 608.453,Z 609.791,A -85,B 0,C 180,E1 -457.801,E2 -457.801} C_VEL
LIN {X 0,Y 608.473,Z 600.815,A -85,B 0,C 180,E1 -458.972,E2 -458.972} C_VEL
LIN {X 0,Y 608.472,Z 591.381,A -85,B 0,C 180,E1 -459.978,E2 -459.978} C_VEL
LIN {X 0,Y 608.506,Z 580.044,A -85,B 0,C 180,E1 -460.973,E2 -460.973} C_VEL
LIN {X 0,Y 608.533,Z 568.134,A -85,B 0,C 180,E1 -461.83,E2 -461.83} C_VEL
LIN {X 0,Y 608.531,Z 555.055,A -85,B 0,C 180,E1 -462.592,E2 -462.592} C_VEL
LIN {X 0,Y 608.556,Z 542.15,A -85,B 0,C 180,E1 -463.185,E2 -463.185} C_VEL
LIN {X 0,Y 608.593,Z 528.15,A -85,B 0,C 180,E1 -463.673,E2 -463.673} C_VEL
LIN {X 0,Y 608.624,Z 514.405,A -85,B 0,C 180,E1 -464.013,E2 -464.013} C_VEL
LIN {X 0,Y 608.622,Z 500.053,A -85,B 0,C 180,E1 -464.235,E2 -464.235} C_VEL
LIN {X 0,Y 608.523,Z 371.979,A -85,B 0,C 180,E1 -465.77,E2 -465.77} C_VEL
LIN {X 0,Y 608.544,Z 348.988,A -85,B 0,C 180,E1 -468.736,E2 -468.736} C_VEL
LIN {X 0,Y 608.563,Z 327.835,A -85,B 0,C 180,E1 -471.511,E2 -471.511} C_VEL
LIN {X 0,Y 608.401,Z 318.321,A -85,B 0,C 180,E1 -472.79,E2 -472.79} C_VEL
LIN {X 0,Y 608.414,Z 318.321,A -85,B 0,C 180,E1 -475.303,E2 -475.303} C_VEL
LIN {X 0,Y 608.418,Z 318.319,A -85,B 0,C 180,E1 -478.269,E2 -478.269} C_VEL
LIN {X 0,Y 608.42,Z 318.317,A -85,B 0,C 180,E1 -480.548,E2 -480.548} C_VEL
LIN {X 0,Y 608.442,Z 318.317,A -85,B 0,C 180,E1 -482.881,E2 -482.881} C_VEL
LIN {X 0,Y 608.437,Z 318.325,A -85,B 0,C 180,E1 -485.279,E2 -485.279} C_VEL
LIN {X 0,Y 608.467,Z 318.313,A -85,B 0,C 180,E1 -487.747,E2 -487.747} C_VEL
LIN {X 0,Y 608.437,Z 318.316,A -85,B 0,C 180,E1 -490.327,E2 -490.327} C_VEL
LIN {X 0,Y 608.456,Z 318.322,A -85,B 0,C 180,E1 -492.96,E2 -492.96} C_VEL
LIN {X 0,Y 608.46,Z 318.312,A -85,B 0,C 180,E1 -495.736,E2 -495.736} C_VEL
LIN {X 0,Y 608.461,Z 318.322,A -85,B 0,C 180,E1 -498.659,E2 -498.659} C_VEL
LIN {X 0,Y 608.468,Z 318.312,A -85,B 0,C 180,E1 -501.76,E2 -501.76} C_VEL
LIN {X 0,Y 608.441,Z 318.319,A -85,B 0,C 180,E1 -504.722,E2 -504.722} C_VEL
LIN {X 0,Y 608.46,Z 318.313,A -85,B 0,C 180,E1 -507.479,E2 -507.479} C_VEL
LIN {X 0,Y 608.474,Z 318.319,A -85,B 0,C 180,E1 -510.221,E2 -510.221} C_VEL
LIN {X 0,Y 608.422,Z 318.317,A -85,B 0,C 180,E1 -512.804,E2 -512.804} C_VEL
LIN {X 0,Y 608.441,Z 318.318,A -85,B 0,C 180,E1 -515.428,E2 -515.428} C_VEL
LIN {X 0,Y 608.431,Z 318.319,A -85,B 0,C 180,E1 -518.307,E2 -518.307} C_VEL
LIN {X 0,Y 608.428,Z 318.37,A -85,B 0,C 180,E1 -518.929,E2 -518.929} C_VEL
LIN {X 0,Y 608.515,Z 333.892,A -85,B 0,C 180,E1 -521.273,E2 -521.273} C_VEL
LIN {X 0,Y 608.484,Z 352.79,A -85,B 0,C 180,E1 -524.079,E2 -524.079} C_VEL
LIN {X 0,Y 608.492,Z 372.626,A -85,B 0,C 180,E1 -526.984,E2 -526.984} C_VEL
LIN {X 0,Y 608.522,Z 373.323,A -85,B 0,C 180,E1 -527.038,E2 -527.038} C_VEL
LIN {X 0,Y 608.554,Z 480.286,A -85,B 0,C 180,E1 -528.319,E2 -528.319} C_VEL
LIN {X 0,Y 608.537,Z 493.618,A -85,B 0,C 180,E1 -528.614,E2 -528.614} C_VEL
LIN {X 0,Y 608.525,Z 506.904,A -85,B 0,C 180,E1 -529.057,E2 -529.057} C_VEL
LIN {X 0,Y 608.504,Z 518.87,A -85,B 0,C 180,E1 -529.603,E2 -529.603} C_VEL
LIN {X 0,Y 608.495,Z 530.292,A -85,B 0,C 180,E1 -530.275,E2 -530.275} C_VEL
LIN {X 0,Y 608.474,Z 540.584,A -85,B 0,C 180,E1 -531.029,E2 -531.029} C_VEL
LIN {X 0,Y 608.464,Z 549.85,A -85,B 0,C 180,E1 -531.866,E2 -531.866} C_VEL
LIN {X 0,Y 608.467,Z 558.824,A -85,B 0,C 180,E1 -532.867,E2 -532.867} C_VEL
LIN {X 0,Y 608.444,Z 566.056,A -85,B 0,C 180,E1 -533.867,E2 -533.867} C_VEL
LIN {X 0,Y 608.462,Z 570.934,A -85,B 0,C 180,E1 -534.698,E2 -534.698} C_VEL
LIN {X 0,Y 608.439,Z 575.679,A -85,B 0,C 180,E1 -535.694,E2 -535.694} C_VEL
LIN {X 0,Y 608.426,Z 579.312,A -85,B 0,C 180,E1 -536.689,E2 -536.689} C_VEL
LIN {X 0,Y 608.425,Z 581.191,A -85,B 0,C 180,E1 -537.352,E2 -537.352} C_VEL
LIN {X 0,Y 608.442,Z 582.626,A -85,B 0,C 180,E1 -538.014,E2 -538.014} C_VEL
LIN {X 0,Y 608.439,Z 584.252,A -85,B 0,C 180,E1 -539.338,E2 -539.338} C_VEL
LIN {X 0,Y 608.434,Z 584.495,A -85,B 0,C 180,E1 -540,E2 -540} C_VEL
LIN {X 0,Y 608.439,Z 584.315,A -85,B 0,C 180,E1 -540.662,E2 -540.662} C_VEL
LIN {X 0,Y 608.441,Z 582.776,A -85,B 0,C 180,E1 -541.986,E2 -541.986} C_VEL
LIN {X 0,Y 608.426,Z 581.418,A -85,B 0,C 180,E1 -542.648,E2 -542.648} C_VEL
LIN {X 0,Y 608.45,Z 578.541,A -85,B 0,C 180,E1 -543.642,E2 -543.642} C_VEL
LIN {X 0,Y 608.433,Z 574.643,A -85,B 0,C 180,E1 -544.638,E2 -544.638} C_VEL
LIN {X 0,Y 608.449,Z 569.611,A -85,B 0,C 180,E1 -545.634,E2 -545.634} C_VEL
LIN {X 0,Y 608.442,Z 563.294,A -85,B 0,C 180,E1 -546.633,E2 -546.633} C_VEL
LIN {X 0,Y 608.475,Z 555.379,A -85,B 0,C 180,E1 -547.633,E2 -547.633} C_VEL
LIN {X 0,Y 608.472,Z 545.531,A -85,B 0,C 180,E1 -548.636,E2 -548.636} C_VEL
LIN {X 0,Y 608.477,Z 543.429,A -85,B 0,C 180,E1 -548.82,E2 -548.82} C_VEL
LIN {X 0,Y 607.81,Z 539.092,A -85,B 0,C 180,E1 -549.19,E2 -549.19} C_VEL
LIN {X 0,Y 604.968,Z 531.848,A -85,B 0,C 180,E1 -549.77,E2 -549.77} C_VEL
LIN {X 0,Y 602.15,Z 524.201,A -85,B 0,C 180,E1 -550.302,E2 -550.302} C_VEL
LIN {X 0,Y 601.522,Z 519.14,A -85,B 0,C 180,E1 -550.595,E2 -550.595} C_VEL
LIN {X 0,Y 601.547,Z 508.508,A -85,B 0,C 180,E1 -551.096,E2 -551.096} C_VEL
LIN {X 0,Y 601.569,Z 496.078,A -85,B 0,C 180,E1 -551.541,E2 -551.541} C_VEL
LIN {X 0,Y 601.609,Z 482.867,A -85,B 0,C 180,E1 -551.861,E2 -551.861} C_VEL
LIN {X 0,Y 601.618,Z 462.255,A -85,B 0,C 180,E1 -552.138,E2 -552.138} C_VEL
LIN {X 0,Y 601.512,Z 373.496,A -85,B 0,C 180,E1 -553.204,E2 -553.204} C_VEL
LIN {X 0,Y 601.457,Z 372.948,A -85,B 0,C 180,E1 -553.214,E2 -553.214} C_VEL
LIN {X 0,Y 601.472,Z 353.396,A -85,B 0,C 180,E1 -556.112,E2 -556.112} C_VEL
LIN {X 0,Y 601.527,Z 335.18,A -85,B 0,C 180,E1 -558.848,E2 -558.848} C_VEL
LIN {X 0,Y 601.58,Z 321.346,A -85,B 0,C 180,E1 -560.956,E2 -560.956} C_VEL
LIN {X 0,Y 601.445,Z 319.189,A -85,B 0,C 180,E1 -561.328,E2 -561.328} C_VEL
LIN {X 0,Y 601.436,Z 319.197,A -85,B 0,C 180,E1 -564.291,E2 -564.291} C_VEL
LIN {X 0,Y 601.447,Z 319.186,A -85,B 0,C 180,E1 -567.111,E2 -567.111} C_VEL
LIN {X 0,Y 601.433,Z 319.197,A -85,B 0,C 180,E1 -570.164,E2 -570.164} C_VEL
LIN {X 0,Y 601.414,Z 319.191,A -85,B 0,C 180,E1 -572.713,E2 -572.713} C_VEL
LIN {X 0,Y 601.388,Z 319.193,A -85,B 0,C 180,E1 -575.11,E2 -575.11} C_VEL
LIN {X 0,Y 601.437,Z 319.189,A -85,B 0,C 180,E1 -577.419,E2 -577.419} C_VEL
LIN {X 0,Y 601.406,Z 319.199,A -85,B 0,C 180,E1 -579.996,E2 -579.996} C_VEL
LIN {X 0,Y 601.38,Z 319.194,A -85,B 0,C 180,E1 -582.673,E2 -582.673} C_VEL
LIN {X 0,Y 601.403,Z 319.191,A -85,B 0,C 180,E1 -584.532,E2 -584.532} C_VEL
LIN {X 0,Y 601.416,Z 319.195,A -85,B 0,C 180,E1 -587.409,E2 -587.409} C_VEL
LIN {X 0,Y 601.398,Z 319.195,A -85,B 0,C 180,E1 -590.003,E2 -590.003} C_VEL
LIN {X 0,Y 601.392,Z 319.192,A -85,B 0,C 180,E1 -592.624,E2 -592.624} C_VEL
LIN {X 0,Y 601.413,Z 319.194,A -85,B 0,C 180,E1 -595.067,E2 -595.067} C_VEL
LIN {X 0,Y 601.421,Z 319.197,A -85,B 0,C 180,E1 -597.483,E2 -597.483} C_VEL
LIN {X 0,Y 601.373,Z 319.197,A -85,B 0,C 180,E1 -599.861,E2 -599.861} C_VEL
LIN {X 0,Y 601.353,Z 319.197,A -85,B 0,C 180,E1 -602.128,E2 -602.128} C_VEL
LIN {X 0,Y 601.351,Z 319.198,A -85,B 0,C 180,E1 -604.378,E2 -604.378} C_VEL
LIN {X 0,Y 601.402,Z 319.2,A -85,B 0,C 180,E1 -607.316,E2 -607.316} C_VEL
LIN {X 0,Y 601.372,Z 319.219,A -85,B 0,C 180,E1 -608.084,E2 -608.084} C_VEL
LIN {X 0,Y 601.615,Z 326.746,A -85,B 0,C 180,E1 -609.156,E2 -609.156} C_VEL
LIN {X 0,Y 601.563,Z 346.887,A -85,B 0,C 180,E1 -611.964,E2 -611.964} C_VEL
LIN {X 0,Y 601.494,Z 362.313,A -85,B 0,C 180,E1 -614.084,E2 -614.084} C_VEL
LIN {X 0,Y 601.844,Z 367.207,A -85,B 0,C 180,E1 -614.159,E2 -614.159} C_VEL
LIN {X 0,Y 601.732,Z 498.883,A -85,B 0,C 180,E1 -615.766,E2 -615.766} C_VEL
LIN {X 0,Y 601.714,Z 512.925,A -85,B 0,C 180,E1 -616.064,E2 -616.064} C_VEL
LIN {X 0,Y 601.665,Z 527.635,A -85,B 0,C 180,E1 -616.532,E2 -616.532} C_VEL
LIN {X 0,Y 601.609,Z 540.672,A -85,B 0,C 180,E1 -617.089,E2 -617.089} C_VEL
LIN {X 0,Y 601.547,Z 553.334,A -85,B 0,C 180,E1 -617.774,E2 -617.774} C_VEL
LIN {X 0,Y 601.506,Z 564.853,A -85,B 0,C 180,E1 -618.542,E2 -618.542} C_VEL
LIN {X 0,Y 601.482,Z 575.415,A -85,B 0,C 180,E1 -619.394,E2 -619.394} C_VEL
LIN {X 0,Y 601.431,Z 585.897,A -85,B 0,C 180,E1 -620.414,E2 -620.414} C_VEL
LIN {X 0,Y 601.406,Z 594.539,A -85,B 0,C 180,E1 -621.43,E2 -621.43} C_VEL
LIN {X 0,Y 601.392,Z 602.837,A -85,B 0,C 180,E1 -622.613,E2 -622.613} C_VEL
LIN {X 0,Y 601.361,Z 608.512,A -85,B 0,C 180,E1 -623.605,E2 -623.605} C_VEL
LIN {X 0,Y 601.353,Z 613.377,A -85,B 0,C 180,E1 -624.634,E2 -624.634} C_VEL
LIN {X 0,Y 601.345,Z 618.299,A -85,B 0,C 180,E1 -625.978,E2 -625.978} C_VEL
LIN {X 0,Y 601.324,Z 621.731,A -85,B 0,C 180,E1 -627.319,E2 -627.319} C_VEL
LIN {X 0,Y 601.346,Z 623.772,A -85,B 0,C 180,E1 -628.66,E2 -628.66} C_VEL
LIN {X 0,Y 601.334,Z 624.495,A -85,B 0,C 180,E1 -629.999,E2 -629.999} C_VEL
LIN {X 0,Y 601.342,Z 623.879,A -85,B 0,C 180,E1 -631.338,E2 -631.338} C_VEL
LIN {X 0,Y 601.321,Z 621.926,A -85,B 0,C 180,E1 -632.679,E2 -632.679} C_VEL
LIN {X 0,Y 601.346,Z 618.589,A -85,B 0,C 180,E1 -634.02,E2 -634.02} C_VEL
LIN {X 0,Y 601.355,Z 613.766,A -85,B 0,C 180,E1 -635.364,E2 -635.364} C_VEL
LIN {X 0,Y 601.355,Z 607.3,A -85,B 0,C 180,E1 -636.71,E2 -636.71} C_VEL
LIN {X 0,Y 601.399,Z 600.097,A -85,B 0,C 180,E1 -637.891,E2 -637.891} C_VEL
LIN {X 0,Y 601.429,Z 591.205,A -85,B 0,C 180,E1 -639.075,E2 -639.075} C_VEL
LIN {X 0,Y 601.439,Z 581.868,A -85,B 0,C 180,E1 -640.094,E2 -640.094} C_VEL
LIN {X 0,Y 601.504,Z 571.247,A -85,B 0,C 180,E1 -641.049,E2 -641.049} C_VEL
LIN {X 0,Y 601.544,Z 560.113,A -85,B 0,C 180,E1 -641.882,E2 -641.882} C_VEL
LIN {X 0,Y 601.561,Z 547.494,A -85,B 0,C 180,E1 -642.652,E2 -642.652} C_VEL
LIN {X 0,Y 601.626,Z 535.227,A -85,B 0,C 180,E1 -643.252,E2 -643.252} C_VEL
LIN {X 0,Y 601.693,Z 521.18,A -85,B 0,C 180,E1 -643.782,E2 -643.782} C_VEL
LIN {X 0,Y 601.727,Z 507.52,A -85,B 0,C 180,E1 -644.154,E2 -644.154} C_VEL
LIN {X 0,Y 601.744,Z 493.654,A -85,B 0,C 180,E1 -644.4,E2 -644.4} C_VEL
LIN {X 0,Y 601.721,Z 363.65,A -85,B 0,C 180,E1 -645.978,E2 -645.978} C_VEL
LIN {X 0,Y 601.497,Z 362.19,A -85,B 0,C 180,E1 -646.023,E2 -646.023} C_VEL
LIN {X 0,Y 601.531,Z 343.31,A -85,B 0,C 180,E1 -648.622,E2 -648.622} C_VEL
LIN {X 0,Y 601.632,Z 324.642,A -85,B 0,C 180,E1 -651.23,E2 -651.23} C_VEL
LIN {X 0,Y 601.392,Z 319.196,A -85,B 0,C 180,E1 -652.024,E2 -652.024} C_VEL
LIN {X 0,Y 601.381,Z 319.202,A -85,B 0,C 180,E1 -654.878,E2 -654.878} C_VEL
LIN {X 0,Y 601.388,Z 319.197,A -85,B 0,C 180,E1 -657.357,E2 -657.357} C_VEL
LIN {X 0,Y 601.367,Z 319.199,A -85,B 0,C 180,E1 -659.394,E2 -659.394} C_VEL
LIN {X 0,Y 601.374,Z 319.195,A -85,B 0,C 180,E1 -661.727,E2 -661.727} C_VEL
LIN {X 0,Y 601.401,Z 319.191,A -85,B 0,C 180,E1 -664.118,E2 -664.118} C_VEL
LIN {X 0,Y 601.39,Z 319.197,A -85,B 0,C 180,E1 -666.582,E2 -666.582} C_VEL
LIN {X 0,Y 601.383,Z 319.195,A -85,B 0,C 180,E1 -669.529,E2 -669.529} C_VEL
LIN {X 0,Y 601.386,Z 319.193,A -85,B 0,C 180,E1 -671.766,E2 -671.766} C_VEL
LIN {X 0,Y 601.388,Z 319.197,A -85,B 0,C 180,E1 -674.531,E2 -674.531} C_VEL
LIN {X 0,Y 601.418,Z 319.192,A -85,B 0,C 180,E1 -676.426,E2 -676.426} C_VEL
LIN {X 0,Y 601.375,Z 319.196,A -85,B 0,C 180,E1 -679.429,E2 -679.429} C_VEL
LIN {X 0,Y 601.344,Z 319.197,A -85,B 0,C 180,E1 -681.726,E2 -681.726} C_VEL
LIN {X 0,Y 601.371,Z 319.194,A -85,B 0,C 180,E1 -683.741,E2 -683.741} C_VEL
LIN {X 0,Y 601.398,Z 319.2,A -85,B 0,C 180,E1 -686.684,E2 -686.684} C_VEL
LIN {X 0,Y 601.383,Z 319.199,A -85,B 0,C 180,E1 -689.056,E2 -689.056} C_VEL
LIN {X 0,Y 601.38,Z 319.195,A -85,B 0,C 180,E1 -691.37,E2 -691.37} C_VEL
LIN {X 0,Y 601.363,Z 319.195,A -85,B 0,C 180,E1 -693.634,E2 -693.634} C_VEL
LIN {X 0,Y 601.381,Z 319.193,A -85,B 0,C 180,E1 -695.856,E2 -695.856} C_VEL
LIN {X 0,Y 601.382,Z 319.203,A -85,B 0,C 180,E1 -698.76,E2 -698.76} C_VEL
LIN {X 0,Y 601.347,Z 319.197,A -85,B 0,C 180,E1 -701.606,E2 -701.606} C_VEL
LIN {X 0,Y 601.372,Z 319.194,A -85,B 0,C 180,E1 -703.711,E2 -703.711} C_VEL
LIN {X 0,Y 601.39,Z 319.2,A -85,B 0,C 180,E1 -706.483,E2 -706.483} C_VEL
LIN {X 0,Y 601.364,Z 319.197,A -85,B 0,C 180,E1 -709.223,E2 -709.223} C_VEL
LIN {X 0,Y 601.377,Z 319.195,A -85,B 0,C 180,E1 -711.938,E2 -711.938} C_VEL
LIN {X 0,Y 601.41,Z 319.2,A -85,B 0,C 180,E1 -714.636,E2 -714.636} C_VEL
LIN {X 0,Y 601.386,Z 319.193,A -85,B 0,C 180,E1 -717.321,E2 -717.321} C_VEL
LIN {X 0,Y 601.4,Z 319.193,A -85,B 0,C 180,E1 -720,E2 -720} C_VEL
LIN {X 0,Y 601.434,Z 319.195,A -85,B 0,C 180,E1 -722.679,E2 -722.679} C_VEL
LIN {X 0,Y 601.369,Z 319.195,A -85,B 0,C 180,E1 -725.365,E2 -725.365} C_VEL
LIN {X 0,Y 601.348,Z 319.197,A -85,B 0,C 180,E1 -727.386,E2 -727.386} C_VEL
LIN {X 0,Y 601.374,Z 319.198,A -85,B 0,C 180,E1 -730.096,E2 -730.096} C_VEL
LIN {X 0,Y 601.389,Z 319.197,A -85,B 0,C 180,E1 -732.829,E2 -732.829} C_VEL
LIN {X 0,Y 601.361,Z 319.196,A -85,B 0,C 180,E1 -735.593,E2 -735.593} C_VEL
LIN {X 0,Y 601.394,Z 319.202,A -85,B 0,C 180,E1 -738.393,E2 -738.393} C_VEL
LIN {X 0,Y 601.367,Z 319.195,A -85,B 0,C 180,E1 -741.241,E2 -741.241} C_VEL
LIN {X 0,Y 601.428,Z 319.193,A -85,B 0,C 180,E1 -744.142,E2 -744.142} C_VEL
LIN {X 0,Y 601.363,Z 319.196,A -85,B 0,C 180,E1 -747.115,E2 -747.115} C_VEL
LIN {X 0,Y 601.359,Z 319.195,A -85,B 0,C 180,E1 -749.396,E2 -749.396} C_VEL
LIN {X 0,Y 601.42,Z 319.196,A -85,B 0,C 180,E1 -752.516,E2 -752.516} C_VEL
LIN {X 0,Y 601.346,Z 319.198,A -85,B 0,C 180,E1 -755.108,E2 -755.108} C_VEL
LIN {X 0,Y 601.369,Z 319.195,A -85,B 0,C 180,E1 -757.424,E2 -757.424} C_VEL
LIN {X 0,Y 601.379,Z 319.199,A -85,B 0,C 180,E1 -759.998,E2 -759.998} C_VEL
LIN {X 0,Y 601.365,Z 319.199,A -85,B 0,C 180,E1 -762.674,E2 -762.674} C_VEL
LIN {X 0,Y 601.353,Z 319.197,A -85,B 0,C 180,E1 -765.477,E2 -765.477} C_VEL
LIN {X 0,Y 601.391,Z 319.199,A -85,B 0,C 180,E1 -768.41,E2 -768.41} C_VEL
LIN {X 0,Y 601.367,Z 319.196,A -85,B 0,C 180,E1 -770.872,E2 -770.872} C_VEL
LIN {X 0,Y 601.374,Z 319.198,A -85,B 0,C 180,E1 -773.743,E2 -773.743} C_VEL
LIN {X 0,Y 601.371,Z 319.197,A -85,B 0,C 180,E1 -776.685,E2 -776.685} C_VEL
LIN {X 0,Y 601.372,Z 319.194,A -85,B 0,C 180,E1 -779.057,E2 -779.057} C_VEL
LIN {X 0,Y 601.35,Z 319.198,A -85,B 0,C 180,E1 -781.37,E2 -781.37} C_VEL
LIN {X 0,Y 601.394,Z 319.198,A -85,B 0,C 180,E1 -784.382,E2 -784.382} C_VEL
LIN {X 0,Y 601.376,Z 319.197,A -85,B 0,C 180,E1 -786.954,E2 -786.954} C_VEL
LIN {X 0,Y 601.389,Z 319.459,A -85,B 0,C 180,E1 -787.09,E2 -787.09} C_VEL
LIN {X 0,Y 601.665,Z 326.509,A -85,B 0,C 180,E1 -788.052,E2 -788.052} C_VEL
LIN {X 0,Y 601.599,Z 347.993,A -85,B 0,C 180,E1 -790.908,E2 -790.908} C_VEL
LIN {X 0,Y 601.52,Z 370.82,A -85,B 0,C 180,E1 -793.891,E2 -793.891} C_VEL
LIN {X 0,Y 601.521,Z 371.953,A -85,B 0,C 180,E1 -794.038,E2 -794.038} C_VEL
LIN {X 0,Y 601.853,Z 375.717,A -85,B 0,C 180,E1 -794.096,E2 -794.096} C_VEL
LIN {X 0,Y 601.753,Z 508.982,A -85,B 0,C 180,E1 -795.722,E2 -795.722} C_VEL
LIN {X 0,Y 601.713,Z 523.29,A -85,B 0,C 180,E1 -796.029,E2 -796.029} C_VEL
LIN {X 0,Y 601.65,Z 537.741,A -85,B 0,C 180,E1 -796.491,E2 -796.491} C_VEL
LIN {X 0,Y 601.608,Z 551.658,A -85,B 0,C 180,E1 -797.091,E2 -797.091} C_VEL
LIN {X 0,Y 601.546,Z 564.113,A -85,B 0,C 180,E1 -797.776,E2 -797.776} C_VEL
LIN {X 0,Y 601.503,Z 575.488,A -85,B 0,C 180,E1 -798.544,E2 -798.544} C_VEL
LIN {X 0,Y 601.481,Z 585.945,A -85,B 0,C 180,E1 -799.397,E2 -799.397} C_VEL
LIN {X 0,Y 601.43,Z 596.345,A -85,B 0,C 180,E1 -800.416,E2 -800.416} C_VEL
LIN {X 0,Y 601.406,Z 604.922,A -85,B 0,C 180,E1 -801.432,E2 -801.432} C_VEL
LIN {X 0,Y 601.391,Z 613.121,A -85,B 0,C 180,E1 -802.615,E2 -802.615} C_VEL
LIN {X 0,Y 601.361,Z 618.752,A -85,B 0,C 180,E1 -803.605,E2 -803.605} C_VEL
LIN {X 0,Y 601.355,Z 623.572,A -85,B 0,C 180,E1 -804.636,E2 -804.636} C_VEL
LIN {X 0,Y 601.343,Z 628.445,A -85,B 0,C 180,E1 -805.98,E2 -805.98} C_VEL
LIN {X 0,Y 601.324,Z 631.834,A -85,B 0,C 180,E1 -807.321,E2 -807.321} C_VEL
LIN {X 0,Y 601.342,Z 633.832,A -85,B 0,C 180,E1 -808.662,E2 -808.662} C_VEL
LIN {X 0,Y 601.333,Z 634.5,A -85,B 0,C 180,E1 -810.001,E2 -810.001} C_VEL
LIN {X 0,Y 601.342,Z 633.83,A -85,B 0,C 180,E1 -811.34,E2 -811.34} C_VEL
LIN {X 0,Y 601.324,Z 631.829,A -85,B 0,C 180,E1 -812.681,E2 -812.681} C_VEL
LIN {X 0,Y 601.343,Z 628.438,A -85,B 0,C 180,E1 -814.022,E2 -814.022} C_VEL
LIN {X 0,Y 601.355,Z 623.564,A -85,B 0,C 180,E1 -815.366,E2 -815.366} C_VEL
LIN {X 0,Y 601.356,Z 617.046,A -85,B 0,C 180,E1 -816.712,E2 -816.712} C_VEL
LIN {X 0,Y 601.398,Z 609.792,A -85,B 0,C 180,E1 -817.893,E2 -817.893} C_VEL
LIN {X 0,Y 601.43,Z 600.815,A -85,B 0,C 180,E1 -819.077,E2 -819.077} C_VEL
LIN {X 0,Y 601.44,Z 591.381,A -85,B 0,C 180,E1 -820.096,E2 -820.096} C_VEL
LIN {X 0,Y 601.506,Z 580.689,A -85,B 0,C 180,E1 -821.051,E2 -821.051} C_VEL
LIN {X 0,Y 601.545,Z 569.413,A -85,B 0,C 180,E1 -821.884,E2 -821.884} C_VEL
LIN {X 0,Y 601.565,Z 556.627,A -85,B 0,C 180,E1 -822.654,E2 -822.654} C_VEL
LIN {X 0,Y 601.626,Z 544.139,A -85,B 0,C 180,E1 -823.254,E2 -823.254} C_VEL
LIN {X 0,Y 601.691,Z 530.817,A -85,B 0,C 180,E1 -823.749,E2 -823.749} C_VEL
LIN {X 0,Y 601.702,Z 516.474,A -85,B 0,C 180,E1 -824.136,E2 -824.136} C_VEL
LIN {X 0,Y 601.746,Z 502.019,A -85,B 0,C 180,E1 -824.377,E2 -824.377} C_VEL
LIN {X 0,Y 601.727,Z 373.209,A -85,B 0,C 180,E1 -825.938,E2 -825.938} C_VEL
LIN {X 0,Y 601.539,Z 371.811,A -85,B 0,C 180,E1 -825.98,E2 -825.98} C_VEL
LIN {X 0,Y 601.583,Z 349.718,A -85,B 0,C 180,E1 -828.865,E2 -828.865} C_VEL
LIN {X 0,Y 601.683,Z 327.835,A -85,B 0,C 180,E1 -831.769,E2 -831.769} C_VEL
LIN {X 0,Y 601.464,Z 319.779,A -85,B 0,C 180,E1 -832.863,E2 -832.863} C_VEL
LIN {X 0,Y 601.352,Z 319.202,A -85,B 0,C 180,E1 -832.959,E2 -832.959} C_VEL
LIN {X 0,Y 601.411,Z 319.199,A -85,B 0,C 180,E1 -835.619,E2 -835.619} C_VEL
LIN {X 0,Y 601.367,Z 319.196,A -85,B 0,C 180,E1 -838.631,E2 -838.631} C_VEL
LIN {X 0,Y 601.418,Z 319.199,A -85,B 0,C 180,E1 -841.454,E2 -841.454} C_VEL
LIN {X 0,Y 601.422,Z 319.189,A -85,B 0,C 180,E1 -844.12,E2 -844.12} C_VEL
LIN {X 0,Y 601.396,Z 319.193,A -85,B 0,C 180,E1 -846.584,E2 -846.584} C_VEL
LIN {X 0,Y 601.446,Z 319.189,A -85,B 0,C 180,E1 -849.536,E2 -849.536} C_VEL
LIN {X 0,Y 601.409,Z 319.195,A -85,B 0,C 180,E1 -852.59,E2 -852.59} C_VEL
LIN {X 0,Y 601.431,Z 319.189,A -85,B 0,C 180,E1 -855.482,E2 -855.482} C_VEL
LIN {X 0,Y 601.426,Z 319.194,A -85,B 0,C 180,E1 -858.407,E2 -858.407} C_VEL
LIN {X 0,Y 601.403,Z 319.196,A -85,B 0,C 180,E1 -860.873,E2 -860.873} C_VEL
LIN {X 0,Y 601.395,Z 319.192,A -85,B 0,C 180,E1 -863.416,E2 -863.416} C_VEL
LIN {X 0,Y 601.435,Z 319.193,A -85,B 0,C 180,E1 -866.065,E2 -866.065} C_VEL
LIN {X 0,Y 601.418,Z 319.194,A -85,B 0,C 180,E1 -868.547,E2 -868.547} C_VEL
LIN {X 0,Y 601.421,Z 319.19,A -85,B 0,C 180,E1 -871.373,E2 -871.373} C_VEL
LIN {X 0,Y 601.388,Z 319.196,A -85,B 0,C 180,E1 -874.381,E2 -874.381} C_VEL
LIN {X 0,Y 601.369,Z 319.197,A -85,B 0,C 180,E1 -876.588,E2 -876.588} C_VEL
LIN {X 0,Y 601.397,Z 319.375,A -85,B 0,C 180,E1 -878.825,E2 -878.825} C_VEL
LIN {X 0,Y 601.572,Z 331.791,A -85,B 0,C 180,E1 -880.729,E2 -880.729} C_VEL
LIN {X 0,Y 601.494,Z 351.627,A -85,B 0,C 180,E1 -883.715,E2 -883.715} C_VEL
LIN {X 0,Y 601.442,Z 371.463,A -85,B 0,C 180,E1 -886.657,E2 -886.657} C_VEL
LIN {X 0,Y 601.463,Z 372.922,A -85,B 0,C 180,E1 -886.872,E2 -886.872} C_VEL
LIN {X 0,Y 601.647,Z 386.781,A -85,B 0,C 180,E1 -887.048,E2 -887.048} C_VEL
LIN {X 0,Y 601.627,Z 480.301,A -85,B 0,C 180,E1 -888.183,E2 -888.183} C_VEL
LIN {X 0,Y 601.601,Z 493.641,A -85,B 0,C 180,E1 -888.481,E2 -888.481} C_VEL
LIN {X 0,Y 601.54,Z 506.036,A -85,B 0,C 180,E1 -888.894,E2 -888.894} C_VEL
LIN {X 0,Y 601.541,Z 517.242,A -85,B 0,C 180,E1 -889.396,E2 -889.396} C_VEL
LIN {X 0,Y 601.467,Z 527.715,A -85,B 0,C 180,E1 -889.991,E2 -889.991} C_VEL
LIN {X 0,Y 601.433,Z 538.473,A -85,B 0,C 180,E1 -890.754,E2 -890.754} C_VEL
LIN {X 0,Y 601.429,Z 548.14,A -85,B 0,C 180,E1 -891.601,E2 -891.601} C_VEL
LIN {X 0,Y 601.418,Z 556.072,A -85,B 0,C 180,E1 -892.446,E2 -892.446} C_VEL
LIN {X 0,Y 601.377,Z 563.389,A -85,B 0,C 180,E1 -893.393,E2 -893.393} C_VEL
LIN {X 0,Y 601.372,Z 569.111,A -85,B 0,C 180,E1 -894.299,E2 -894.299} C_VEL
LIN {X 0,Y 601.335,Z 574.249,A -85,B 0,C 180,E1 -895.307,E2 -895.307} C_VEL
LIN {X 0,Y 601.368,Z 578.243,A -85,B 0,C 180,E1 -896.315,E2 -896.315} C_VEL
LIN {X 0,Y 601.324,Z 581.193,A -85,B 0,C 180,E1 -897.32,E2 -897.32} C_VEL
LIN {X 0,Y 601.341,Z 582.624,A -85,B 0,C 180,E1 -897.991,E2 -897.991} C_VEL
LIN {X 0,Y 601.339,Z 584.255,A -85,B 0,C 180,E1 -899.33,E2 -899.33} C_VEL
LIN {X 0,Y 601.335,Z 584.496,A -85,B 0,C 180,E1 -900,E2 -900} C_VEL
LIN {X 0,Y 601.339,Z 584.317,A -85,B 0,C 180,E1 -900.67,E2 -900.67} C_VEL
LIN {X 0,Y 601.34,Z 582.773,A -85,B 0,C 180,E1 -902.009,E2 -902.009} C_VEL
LIN {X 0,Y 601.326,Z 581.412,A -85,B 0,C 180,E1 -902.68,E2 -902.68} C_VEL
LIN {X 0,Y 601.368,Z 578.538,A -85,B 0,C 180,E1 -903.685,E2 -903.685} C_VEL
LIN {X 0,Y 601.337,Z 574.644,A -85,B 0,C 180,E1 -904.693,E2 -904.693} C_VEL
LIN {X 0,Y 601.373,Z 569.606,A -85,B 0,C 180,E1 -905.701,E2 -905.701} C_VEL
LIN {X 0,Y 601.383,Z 563.289,A -85,B 0,C 180,E1 -906.711,E2 -906.711} C_VEL
LIN {X 0,Y 601.396,Z 555.377,A -85,B 0,C 180,E1 -907.723,E2 -907.723} C_VEL
LIN {X 0,Y 601.422,Z 547.307,A -85,B 0,C 180,E1 -908.569,E2 -908.569} C_VEL
LIN {X 0,Y 601.453,Z 537.475,A -85,B 0,C 180,E1 -909.415,E2 -909.415} C_VEL
LIN {X 0,Y 601.481,Z 526.417,A -85,B 0,C 180,E1 -910.179,E2 -910.179} C_VEL
LIN {X 0,Y 601.522,Z 519.14,A -85,B 0,C 180,E1 -910.595,E2 -910.595} C_VEL
LIN {X 0,Y 600.883,Z 514.008,A -85,B 0,C 180,E1 -910.869,E2 -910.869} C_VEL
LIN {X 0,Y 598.038,Z 505.555,A -85,B 0,C 180,E1 -911.287,E2 -911.287} C_VEL
LIN {X 0,Y 595.242,Z 496.809,A -85,B 0,C 180,E1 -911.642,E2 -911.642} C_VEL
LIN {X 0,Y 594.632,Z 491.225,A -85,B 0,C 180,E1 -911.814,E2 -911.814} C_VEL
LIN {X 0,Y 594.696,Z 477.771,A -85,B 0,C 180,E1 -912.087,E2 -912.087} C_VEL
LIN {X 0,Y 594.589,Z 374.143,A -85,B 0,C 180,E1 -913.353,E2 -913.353} C_VEL
LIN {X 0,Y 594.403,Z 372.945,A -85,B 0,C 180,E1 -913.374,E2 -913.374} C_VEL
LIN {X 0,Y 594.482,Z 354.559,A -85,B 0,C 180,E1 -916.13,E2 -916.13} C_VEL
LIN {X 0,Y 594.577,Z 335.055,A -85,B 0,C 180,E1 -919.096,E2 -919.096} C_VEL
LIN {X 0,Y 594.563,Z 321.54,A -85,B 0,C 180,E1 -921.184,E2 -921.184} C_VEL
LIN {X 0,Y 594.406,Z 320.067,A -85,B 0,C 180,E1 -921.424,E2 -921.424} C_VEL
LIN {X 0,Y 594.394,Z 320.072,A -85,B 0,C 180,E1 -924.446,E2 -924.446} C_VEL
LIN {X 0,Y 594.382,Z 320.069,A -85,B 0,C 180,E1 -926.7,E2 -926.7} C_VEL
LIN {X 0,Y 594.38,Z 320.066,A -85,B 0,C 180,E1 -928.999,E2 -928.999} C_VEL
LIN {X 0,Y 594.38,Z 320.069,A -85,B 0,C 180,E1 -931.642,E2 -931.642} C_VEL
LIN {X 0,Y 594.374,Z 320.069,A -85,B 0,C 180,E1 -934.581,E2 -934.581} C_VEL
LIN {X 0,Y 594.391,Z 320.069,A -85,B 0,C 180,E1 -937.608,E2 -937.608} C_VEL
LIN {X 0,Y 594.362,Z 320.069,A -85,B 0,C 180,E1 -940.568,E2 -940.568} C_VEL
LIN {X 0,Y 594.363,Z 320.071,A -85,B 0,C 180,E1 -943.3,E2 -943.3} C_VEL
LIN {X 0,Y 594.347,Z 320.073,A -85,B 0,C 180,E1 -946.163,E2 -946.163} C_VEL
LIN {X 0,Y 594.366,Z 320.068,A -85,B 0,C 180,E1 -948.534,E2 -948.534} C_VEL
LIN {X 0,Y 594.368,Z 320.073,A -85,B 0,C 180,E1 -951.298,E2 -951.298} C_VEL
LIN {X 0,Y 594.345,Z 320.076,A -85,B 0,C 180,E1 -953.754,E2 -953.754} C_VEL
LIN {X 0,Y 594.335,Z 320.072,A -85,B 0,C 180,E1 -956.235,E2 -956.235} C_VEL
LIN {X 0,Y 594.342,Z 320.072,A -85,B 0,C 180,E1 -958.647,E2 -958.647} C_VEL
LIN {X 0,Y 594.377,Z 320.073,A -85,B 0,C 180,E1 -961.044,E2 -961.044} C_VEL
LIN {X 0,Y 594.319,Z 320.075,A -85,B 0,C 180,E1 -963.991,E2 -963.991} C_VEL
LIN {X 0,Y 594.326,Z 320.074,A -85,B 0,C 180,E1 -966.292,E2 -966.292} C_VEL
LIN {X 0,Y 594.35,Z 320.177,A -85,B 0,C 180,E1 -967.948,E2 -967.948} C_VEL
LIN {X 0,Y 594.697,Z 326.138,A -85,B 0,C 180,E1 -968.815,E2 -968.815} C_VEL
LIN {X 0,Y 594.578,Z 344.347,A -85,B 0,C 180,E1 -971.388,E2 -971.388} C_VEL
LIN {X 0,Y 594.525,Z 362.317,A -85,B 0,C 180,E1 -973.892,E2 -973.892} C_VEL
LIN {X 0,Y 595.022,Z 367.253,A -85,B 0,C 180,E1 -973.972,E2 -973.972} C_VEL
LIN {X 0,Y 594.867,Z 499.699,A -85,B 0,C 180,E1 -975.612,E2 -975.612} C_VEL
LIN {X 0,Y 594.826,Z 513.711,A -85,B 0,C 180,E1 -975.92,E2 -975.92} C_VEL
LIN {X 0,Y 594.752,Z 527.65,A -85,B 0,C 180,E1 -976.372,E2 -976.372} C_VEL
LIN {X 0,Y 594.663,Z 540.671,A -85,B 0,C 180,E1 -976.936,E2 -976.936} C_VEL
LIN {X 0,Y 594.601,Z 551.92,A -85,B 0,C 180,E1 -977.542,E2 -977.542} C_VEL
LIN {X 0,Y 594.508,Z 563.704,A -85,B 0,C 180,E1 -978.319,E2 -978.319} C_VEL
LIN {X 0,Y 594.474,Z 575.425,A -85,B 0,C 180,E1 -979.268,E2 -979.268} C_VEL
LIN {X 0,Y 594.392,Z 585.896,A -85,B 0,C 180,E1 -980.299,E2 -980.299} C_VEL
LIN {X 0,Y 594.355,Z 594.534,A -85,B 0,C 180,E1 -981.328,E2 -981.328} C_VEL
LIN {X 0,Y 594.315,Z 602.84,A -85,B 0,C 180,E1 -982.525,E2 -982.525} C_VEL
LIN {X 0,Y 594.271,Z 609.005,A -85,B 0,C 180,E1 -983.62,E2 -983.62} C_VEL
LIN {X 0,Y 594.246,Z 614.777,A -85,B 0,C 180,E1 -984.91,E2 -984.91} C_VEL
LIN {X 0,Y 594.261,Z 618.303,A -85,B 0,C 180,E1 -985.93,E2 -985.93} C_VEL
LIN {X 0,Y 594.224,Z 621.731,A -85,B 0,C 180,E1 -987.287,E2 -987.287} C_VEL
LIN {X 0,Y 594.245,Z 623.77,A -85,B 0,C 180,E1 -988.644,E2 -988.644} C_VEL
LIN {X 0,Y 594.235,Z 624.495,A -85,B 0,C 180,E1 -989.999,E2 -989.999} C_VEL
LIN {X 0,Y 594.242,Z 623.875,A -85,B 0,C 180,E1 -991.354,E2 -991.354} C_VEL
LIN {X 0,Y 594.221,Z 621.918,A -85,B 0,C 180,E1 -992.711,E2 -992.711} C_VEL
LIN {X 0,Y 594.262,Z 618.59,A -85,B 0,C 180,E1 -994.068,E2 -994.068} C_VEL
LIN {X 0,Y 594.275,Z 613.767,A -85,B 0,C 180,E1 -995.428,E2 -995.428} C_VEL
LIN {X 0,Y 594.276,Z 607.299,A -85,B 0,C 180,E1 -996.791,E2 -996.791} C_VEL
LIN {X 0,Y 594.329,Z 600.088,A -85,B 0,C 180,E1 -997.986,E2 -997.986} C_VEL
LIN {X 0,Y 594.384,Z 591.199,A -85,B 0,C 180,E1 -999.184,E2 -999.184} C_VEL
LIN {X 0,Y 594.411,Z 581.86,A -85,B 0,C 180,E1 -1000.214,E2 -1000.214} C_VEL
LIN {X 0,Y 594.506,Z 571.864,A -85,B 0,C 180,E1 -1001.13,E2 -1001.13} C_VEL
LIN {X 0,Y 594.57,Z 561.354,A -85,B 0,C 180,E1 -1001.937,E2 -1001.937} C_VEL
LIN {X 0,Y 594.613,Z 550.549,A -85,B 0,C 180,E1 -1002.629,E2 -1002.629} C_VEL
LIN {X 0,Y 594.69,Z 537.191,A -85,B 0,C 180,E1 -1003.322,E2 -1003.322} C_VEL
LIN {X 0,Y 594.786,Z 523.547,A -85,B 0,C 180,E1 -1003.865,E2 -1003.865} C_VEL
LIN {X 0,Y 594.812,Z 509.874,A -85,B 0,C 180,E1 -1004.265,E2 -1004.265} C_VEL
LIN {X 0,Y 594.866,Z 495.801,A -85,B 0,C 180,E1 -1004.539,E2 -1004.539} C_VEL
LIN {X 0,Y 594.97,Z 364.902,A -85,B 0,C 180,E1 -1006.148,E2 -1006.148} C_VEL
LIN {X 0,Y 594.53,Z 362.186,A -85,B 0,C 180,E1 -1006.216,E2 -1006.216} C_VEL
LIN {X 0,Y 594.635,Z 341.513,A -85,B 0,C 180,E1 -1009.099,E2 -1009.099} C_VEL
LIN {X 0,Y 594.709,Z 323.365,A -85,B 0,C 180,E1 -1011.671,E2 -1011.671} C_VEL
LIN {X 0,Y 594.33,Z 320.077,A -85,B 0,C 180,E1 -1012.188,E2 -1012.188} C_VEL
LIN {X 0,Y 594.336,Z 320.074,A -85,B 0,C 180,E1 -1014.447,E2 -1014.447} C_VEL
LIN {X 0,Y 594.361,Z 320.074,A -85,B 0,C 180,E1 -1016.699,E2 -1016.699} C_VEL
LIN {X 0,Y 594.364,Z 320.078,A -85,B 0,C 180,E1 -1018.998,E2 -1018.998} C_VEL
LIN {X 0,Y 594.349,Z 320.071,A -85,B 0,C 180,E1 -1021.638,E2 -1021.638} C_VEL
LIN {X 0,Y 594.371,Z 320.071,A -85,B 0,C 180,E1 -1024.579,E2 -1024.579} C_VEL
LIN {X 0,Y 594.348,Z 320.071,A -85,B 0,C 180,E1 -1027.603,E2 -1027.603} C_VEL
LIN {X 0,Y 594.347,Z 320.074,A -85,B 0,C 180,E1 -1030.567,E2 -1030.567} C_VEL
LIN {X 0,Y 594.332,Z 320.075,A -85,B 0,C 180,E1 -1033.301,E2 -1033.301} C_VEL
LIN {X 0,Y 594.349,Z 320.07,A -85,B 0,C 180,E1 -1036.16,E2 -1036.16} C_VEL
LIN {X 0,Y 594.351,Z 320.074,A -85,B 0,C 180,E1 -1039.179,E2 -1039.179} C_VEL
LIN {X 0,Y 594.338,Z 320.07,A -85,B 0,C 180,E1 -1042.056,E2 -1042.056} C_VEL
LIN {X 0,Y 594.311,Z 320.082,A -85,B 0,C 180,E1 -1044.679,E2 -1044.679} C_VEL
LIN {X 0,Y 594.357,Z 320.073,A -85,B 0,C 180,E1 -1047.089,E2 -1047.089} C_VEL
LIN {X 0,Y 594.334,Z 320.071,A -85,B 0,C 180,E1 -1049.677,E2 -1049.677} C_VEL
LIN {X 0,Y 594.305,Z 320.074,A -85,B 0,C 180,E1 -1051.769,E2 -1051.769} C_VEL
LIN {X 0,Y 594.341,Z 320.07,A -85,B 0,C 180,E1 -1054.054,E2 -1054.054} C_VEL
LIN {X 0,Y 594.332,Z 320.076,A -85,B 0,C 180,E1 -1057.031,E2 -1057.031} C_VEL
LIN {X 0,Y 594.337,Z 320.07,A -85,B 0,C 180,E1 -1059.945,E2 -1059.945} C_VEL
LIN {X 0,Y 594.357,Z 320.077,A -85,B 0,C 180,E1 -1062.806,E2 -1062.806} C_VEL
LIN {X 0,Y 594.314,Z 320.074,A -85,B 0,C 180,E1 -1065.848,E2 -1065.848} C_VEL
LIN {X 0,Y 594.351,Z 320.074,A -85,B 0,C 180,E1 -1068.937,E2 -1068.937} C_VEL
LIN {X 0,Y 594.33,Z 320.072,A -85,B 0,C 180,E1 -1071.842,E2 -1071.842} C_VEL
LIN {X 0,Y 594.371,Z 320.077,A -85,B 0,C 180,E1 -1074.572,E2 -1074.572} C_VEL
LIN {X 0,Y 594.357,Z 320.069,A -85,B 0,C 180,E1 -1077.289,E2 -1077.289} C_VEL
LIN {X 0,Y 594.371,Z 320.068,A -85,B 0,C 180,E1 -1080,E2 -1080} C_VEL
LIN {X 0,Y 594.394,Z 320.071,A -85,B 0,C 180,E1 -1082.711,E2 -1082.711} C_VEL
LIN {X 0,Y 594.336,Z 320.071,A -85,B 0,C 180,E1 -1085.428,E2 -1085.428} C_VEL
LIN {X 0,Y 594.322,Z 320.072,A -85,B 0,C 180,E1 -1087.474,E2 -1087.474} C_VEL
LIN {X 0,Y 594.309,Z 320.074,A -85,B 0,C 180,E1 -1089.53,E2 -1089.53} C_VEL
LIN {X 0,Y 594.358,Z 320.075,A -85,B 0,C 180,E1 -1092.289,E2 -1092.289} C_VEL
LIN {X 0,Y 594.34,Z 320.072,A -85,B 0,C 180,E1 -1095.079,E2 -1095.079} C_VEL
LIN {X 0,Y 594.321,Z 320.073,A -85,B 0,C 180,E1 -1097.195,E2 -1097.195} C_VEL
LIN {X 0,Y 594.336,Z 320.071,A -85,B 0,C 180,E1 -1099.335,E2 -1099.335} C_VEL
LIN {X 0,Y 594.331,Z 320.071,A -85,B 0,C 180,E1 -1101.505,E2 -1101.505} C_VEL
LIN {X 0,Y 594.372,Z 320.076,A -85,B 0,C 180,E1 -1104.447,E2 -1104.447} C_VEL
LIN {X 0,Y 594.327,Z 320.072,A -85,B 0,C 180,E1 -1107.519,E2 -1107.519} C_VEL
LIN {X 0,Y 594.35,Z 320.079,A -85,B 0,C 180,E1 -1110.325,E2 -1110.325} C_VEL
LIN {X 0,Y 594.354,Z 320.07,A -85,B 0,C 180,E1 -1112.952,E2 -1112.952} C_VEL
LIN {X 0,Y 594.296,Z 320.076,A -85,B 0,C 180,E1 -1115.413,E2 -1115.413} C_VEL
LIN {X 0,Y 594.349,Z 320.074,A -85,B 0,C 180,E1 -1117.944,E2 -1117.944} C_VEL
LIN {X 0,Y 594.314,Z 320.076,A -85,B 0,C 180,E1 -1120.817,E2 -1120.817} C_VEL
LIN {X 0,Y 594.328,Z 320.072,A -85,B 0,C 180,E1 -1123.303,E2 -1123.303} C_VEL
LIN {X 0,Y 594.322,Z 320.082,A -85,B 0,C 180,E1 -1126.165,E2 -1126.165} C_VEL
LIN {X 0,Y 594.346,Z 320.075,A -85,B 0,C 180,E1 -1128.535,E2 -1128.535} C_VEL
LIN {X 0,Y 594.315,Z 320.074,A -85,B 0,C 180,E1 -1131.304,E2 -1131.304} C_VEL
LIN {X 0,Y 594.329,Z 320.076,A -85,B 0,C 180,E1 -1133.756,E2 -1133.756} C_VEL
LIN {X 0,Y 594.342,Z 320.08,A -85,B 0,C 180,E1 -1136.238,E2 -1136.238} C_VEL
LIN {X 0,Y 594.345,Z 320.073,A -85,B 0,C 180,E1 -1138.65,E2 -1138.65} C_VEL
LIN {X 0,Y 594.325,Z 320.072,A -85,B 0,C 180,E1 -1141.053,E2 -1141.053} C_VEL
LIN {X 0,Y 594.343,Z 320.079,A -85,B 0,C 180,E1 -1143.986,E2 -1143.986} C_VEL
LIN {X 0,Y 594.363,Z 320.131,A -85,B 0,C 180,E1 -1146.896,E2 -1146.896} C_VEL
LIN {X 0,Y 594.774,Z 325.415,A -85,B 0,C 180,E1 -1147.635,E2 -1147.635} C_VEL
LIN {X 0,Y 594.682,Z 346.65,A -85,B 0,C 180,E1 -1150.498,E2 -1150.498} C_VEL
LIN {X 0,Y 594.545,Z 369.477,A -85,B 0,C 180,E1 -1153.52,E2 -1153.52} C_VEL
LIN {X 0,Y 594.555,Z 372.141,A -85,B 0,C 180,E1 -1153.851,E2 -1153.851} C_VEL
LIN {X 0,Y 595.024,Z 375.717,A -85,B 0,C 180,E1 -1153.908,E2 -1153.908} C_VEL
LIN {X 0,Y 594.855,Z 509.948,A -85,B 0,C 180,E1 -1155.57,E2 -1155.57} C_VEL
LIN {X 0,Y 594.816,Z 524.179,A -85,B 0,C 180,E1 -1155.89,E2 -1155.89} C_VEL
LIN {X 0,Y 594.74,Z 537.742,A -85,B 0,C 180,E1 -1156.331,E2 -1156.331} C_VEL
LIN {X 0,Y 594.663,Z 551.661,A -85,B 0,C 180,E1 -1156.938,E2 -1156.938} C_VEL
LIN {X 0,Y 594.595,Z 564.115,A -85,B 0,C 180,E1 -1157.631,E2 -1157.631} C_VEL
LIN {X 0,Y 594.523,Z 576.573,A -85,B 0,C 180,E1 -1158.489,E2 -1158.489} C_VEL
LIN {X 0,Y 594.448,Z 587.848,A -85,B 0,C 180,E1 -1159.442,E2 -1159.442} C_VEL
LIN {X 0,Y 594.367,Z 597.86,A -85,B 0,C 180,E1 -1160.473,E2 -1160.473} C_VEL
LIN {X 0,Y 594.323,Z 606.178,A -85,B 0,C 180,E1 -1161.501,E2 -1161.501} C_VEL
LIN {X 0,Y 594.302,Z 614.132,A -85,B 0,C 180,E1 -1162.698,E2 -1162.698} C_VEL
LIN {X 0,Y 594.279,Z 620.532,A -85,B 0,C 180,E1 -1163.891,E2 -1163.891} C_VEL
LIN {X 0,Y 594.237,Z 626.203,A -85,B 0,C 180,E1 -1165.252,E2 -1165.252} C_VEL
LIN {X 0,Y 594.259,Z 630.319,A -85,B 0,C 180,E1 -1166.611,E2 -1166.611} C_VEL
LIN {X 0,Y 594.24,Z 633.002,A -85,B 0,C 180,E1 -1167.968,E2 -1167.968} C_VEL
LIN {X 0,Y 594.237,Z 634.333,A -85,B 0,C 180,E1 -1169.323,E2 -1169.323} C_VEL
LIN {X 0,Y 594.237,Z 634.331,A -85,B 0,C 180,E1 -1170.679,E2 -1170.679} C_VEL
LIN {X 0,Y 594.24,Z 632.998,A -85,B 0,C 180,E1 -1172.034,E2 -1172.034} C_VEL
LIN {X 0,Y 594.259,Z 630.313,A -85,B 0,C 180,E1 -1173.391,E2 -1173.391} C_VEL
LIN {X 0,Y 594.237,Z 626.195,A -85,B 0,C 180,E1 -1174.75,E2 -1174.75} C_VEL
LIN {X 0,Y 594.28,Z 620.522,A -85,B 0,C 180,E1 -1176.111,E2 -1176.111} C_VEL
LIN {X 0,Y 594.304,Z 614.12,A -85,B 0,C 180,E1 -1177.304,E2 -1177.304} C_VEL
LIN {X 0,Y 594.324,Z 606.163,A -85,B 0,C 180,E1 -1178.501,E2 -1178.501} C_VEL
LIN {X 0,Y 594.367,Z 597.842,A -85,B 0,C 180,E1 -1179.53,E2 -1179.53} C_VEL
LIN {X 0,Y 594.449,Z 587.827,A -85,B 0,C 180,E1 -1180.56,E2 -1180.56} C_VEL
LIN {X 0,Y 594.525,Z 576.551,A -85,B 0,C 180,E1 -1181.513,E2 -1181.513} C_VEL
LIN {X 0,Y 594.583,Z 564.081,A -85,B 0,C 180,E1 -1182.372,E2 -1182.372} C_VEL
LIN {X 0,Y 594.654,Z 551.618,A -85,B 0,C 180,E1 -1183.064,E2 -1183.064} C_VEL
LIN {X 0,Y 594.74,Z 537.691,A -85,B 0,C 180,E1 -1183.671,E2 -1183.671} C_VEL
LIN {X 0,Y 594.827,Z 523.677,A -85,B 0,C 180,E1 -1184.125,E2 -1184.125} C_VEL
LIN {X 0,Y 594.88,Z 509.839,A -85,B 0,C 180,E1 -1184.431,E2 -1184.431} C_VEL
LIN {X 0,Y 594.973,Z 374.426,A -85,B 0,C 180,E1 -1186.109,E2 -1186.109} C_VEL
LIN {X 0,Y 594.529,Z 371.811,A -85,B 0,C 180,E1 -1186.174,E2 -1186.174} C_VEL
LIN {X 0,Y 594.642,Z 349.645,A -85,B 0,C 180,E1 -1189.103,E2 -1189.103} C_VEL
LIN {X 0,Y 594.768,Z 329.178,A -85,B 0,C 180,E1 -1191.853,E2 -1191.853} C_VEL
LIN {X 0,Y 594.514,Z 321.122,A -85,B 0,C 180,E1 -1192.962,E2 -1192.962} C_VEL
LIN {X 0,Y 594.332,Z 320.078,A -85,B 0,C 180,E1 -1193.153,E2 -1193.153} C_VEL
LIN {X 0,Y 594.357,Z 320.075,A -85,B 0,C 180,E1 -1196.017,E2 -1196.017} C_VEL
LIN {X 0,Y 594.339,Z 320.073,A -85,B 0,C 180,E1 -1199.002,E2 -1199.002} C_VEL
LIN {X 0,Y 594.374,Z 320.074,A -85,B 0,C 180,E1 -1201.642,E2 -1201.642} C_VEL
LIN {X 0,Y 594.369,Z 320.068,A -85,B 0,C 180,E1 -1204.581,E2 -1204.581} C_VEL
LIN {X 0,Y 594.391,Z 320.068,A -85,B 0,C 180,E1 -1207.608,E2 -1207.608} C_VEL
LIN {X 0,Y 594.364,Z 320.071,A -85,B 0,C 180,E1 -1210.568,E2 -1210.568} C_VEL
LIN {X 0,Y 594.37,Z 320.071,A -85,B 0,C 180,E1 -1213.3,E2 -1213.3} C_VEL
LIN {X 0,Y 594.373,Z 320.069,A -85,B 0,C 180,E1 -1216.161,E2 -1216.161} C_VEL
LIN {X 0,Y 594.383,Z 320.074,A -85,B 0,C 180,E1 -1218.536,E2 -1218.536} C_VEL
LIN {X 0,Y 594.375,Z 320.067,A -85,B 0,C 180,E1 -1221.298,E2 -1221.298} C_VEL
LIN {X 0,Y 594.354,Z 320.071,A -85,B 0,C 180,E1 -1223.756,E2 -1223.756} C_VEL
LIN {X 0,Y 594.378,Z 320.075,A -85,B 0,C 180,E1 -1226.239,E2 -1226.239} C_VEL
LIN {X 0,Y 594.367,Z 320.071,A -85,B 0,C 180,E1 -1228.65,E2 -1228.65} C_VEL
LIN {X 0,Y 594.379,Z 320.067,A -85,B 0,C 180,E1 -1231.044,E2 -1231.044} C_VEL
LIN {X 0,Y 594.36,Z 320.077,A -85,B 0,C 180,E1 -1234.055,E2 -1234.055} C_VEL
LIN {X 0,Y 594.363,Z 320.073,A -85,B 0,C 180,E1 -1236.295,E2 -1236.295} C_VEL
LIN {X 0,Y 594.358,Z 320.229,A -85,B 0,C 180,E1 -1238.694,E2 -1238.694} C_VEL
LIN {X 0,Y 594.615,Z 327.128,A -85,B 0,C 180,E1 -1239.774,E2 -1239.774} C_VEL
LIN {X 0,Y 594.515,Z 344.63,A -85,B 0,C 180,E1 -1242.456,E2 -1242.456} C_VEL
LIN {X 0,Y 594.433,Z 363.299,A -85,B 0,C 180,E1 -1245.274,E2 -1245.274} C_VEL
LIN {X 0,Y 594.434,Z 372.925,A -85,B 0,C 180,E1 -1246.714,E2 -1246.714} C_VEL
LIN {X 0,Y 594.763,Z 379.672,A -85,B 0,C 180,E1 -1246.809,E2 -1246.809} C_VEL
LIN {X 0,Y 594.683,Z 480.316,A -85,B 0,C 180,E1 -1248.043,E2 -1248.043} C_VEL
LIN {X 0,Y 594.634,Z 493.664,A -85,B 0,C 180,E1 -1248.344,E2 -1248.344} C_VEL
LIN {X 0,Y 594.56,Z 506.816,A -85,B 0,C 180,E1 -1248.792,E2 -1248.792} C_VEL
LIN {X 0,Y 594.521,Z 518.895,A -85,B 0,C 180,E1 -1249.356,E2 -1249.356} C_VEL
LIN {X 0,Y 594.46,Z 530.316,A -85,B 0,C 180,E1 -1250.043,E2 -1250.043} C_VEL
LIN {X 0,Y 594.406,Z 540.586,A -85,B 0,C 180,E1 -1250.815,E2 -1250.815} C_VEL
LIN {X 0,Y 594.373,Z 549.859,A -85,B 0,C 180,E1 -1251.672,E2 -1251.672} C_VEL
LIN {X 0,Y 594.317,Z 558.834,A -85,B 0,C 180,E1 -1252.697,E2 -1252.697} C_VEL
LIN {X 0,Y 594.285,Z 565.362,A -85,B 0,C 180,E1 -1253.613,E2 -1253.613} C_VEL
LIN {X 0,Y 594.289,Z 570.937,A -85,B 0,C 180,E1 -1254.571,E2 -1254.571} C_VEL
LIN {X 0,Y 594.27,Z 575.689,A -85,B 0,C 180,E1 -1255.591,E2 -1255.591} C_VEL
LIN {X 0,Y 594.268,Z 579.312,A -85,B 0,C 180,E1 -1256.61,E2 -1256.61} C_VEL
LIN {X 0,Y 594.225,Z 581.192,A -85,B 0,C 180,E1 -1257.288,E2 -1257.288} C_VEL
LIN {X 0,Y 594.24,Z 582.621,A -85,B 0,C 180,E1 -1257.967,E2 -1257.967} C_VEL
LIN {X 0,Y 594.24,Z 584.258,A -85,B 0,C 180,E1 -1259.322,E2 -1259.322} C_VEL
LIN {X 0,Y 594.236,Z 584.496,A -85,B 0,C 180,E1 -1260,E2 -1260} C_VEL
LIN {X 0,Y 594.24,Z 584.319,A -85,B 0,C 180,E1 -1260.678,E2 -1260.678} C_VEL
LIN {X 0,Y 594.239,Z 582.771,A -85,B 0,C 180,E1 -1262.033,E2 -1262.033} C_VEL
LIN {X 0,Y 594.226,Z 581.405,A -85,B 0,C 180,E1 -1262.712,E2 -1262.712} C_VEL
LIN {X 0,Y 594.289,Z 578.535,A -85,B 0,C 180,E1 -1263.729,E2 -1263.729} C_VEL
LIN {X 0,Y 594.242,Z 574.644,A -85,B 0,C 180,E1 -1264.749,E2 -1264.749} C_VEL
LIN {X 0,Y 594.299,Z 569.599,A -85,B 0,C 180,E1 -1265.769,E2 -1265.769} C_VEL
LIN {X 0,Y 594.317,Z 563.284,A -85,B 0,C 180,E1 -1266.791,E2 -1266.791} C_VEL
LIN {X 0,Y 594.347,Z 555.375,A -85,B 0,C 180,E1 -1267.816,E2 -1267.816} C_VEL
LIN {X 0,Y 594.366,Z 547.301,A -85,B 0,C 180,E1 -1268.671,E2 -1268.671} C_VEL
LIN {X 0,Y 594.416,Z 537.468,A -85,B 0,C 180,E1 -1269.528,E2 -1269.528} C_VEL
LIN {X 0,Y 594.465,Z 526.412,A -85,B 0,C 180,E1 -1270.301,E2 -1270.301} C_VEL
LIN {X 0,Y 594.538,Z 514.131,A -85,B 0,C 180,E1 -1270.974,E2 -1270.974} C_VEL
LIN {X 0,Y 594.584,Z 502.478,A -85,B 0,C 180,E1 -1271.464,E2 -1271.464} C_VEL
LIN {X 0,Y 594.632,Z 491.225,A -85,B 0,C 180,E1 -1271.814,E2 -1271.814} C_VEL
LIN {X 0,Y 594.044,Z 485.551,A -85,B 0,C 180,E1 -1271.961,E2 -1271.961} C_VEL
LIN {X 0,Y 588.866,Z 468.871,A -85,B 0,C 180,E1 -1272.326,E2 -1272.326} C_VEL
LIN {X 0,Y 587.853,Z 463.116,A -85,B 0,C 180,E1 -1272.416,E2 -1272.416} C_VEL
LIN {X 0,Y 587.779,Z 461.163,A -85,B 0,C 180,E1 -1272.441,E2 -1272.441} C_VEL
LIN {X 0,Y 587.7,Z 374.994,A -85,B 0,C 180,E1 -1273.501,E2 -1273.501} C_VEL
LIN {X 0,Y 587.389,Z 372.941,A -85,B 0,C 180,E1 -1273.536,E2 -1273.536} C_VEL
LIN {X 0,Y 587.473,Z 354.555,A -85,B 0,C 180,E1 -1276.328,E2 -1276.328} C_VEL
LIN {X 0,Y 587.619,Z 335.389,A -85,B 0,C 180,E1 -1279.278,E2 -1279.278} C_VEL
LIN {X 0,Y 587.557,Z 321.87,A -85,B 0,C 180,E1 -1281.396,E2 -1281.396} C_VEL
LIN {X 0,Y 587.369,Z 320.945,A -85,B 0,C 180,E1 -1281.588,E2 -1281.588} C_VEL
LIN {X 0,Y 587.355,Z 320.944,A -85,B 0,C 180,E1 -1284.759,E2 -1284.759} C_VEL
LIN {X 0,Y 587.346,Z 320.945,A -85,B 0,C 180,E1 -1287.691,E2 -1287.691} C_VEL
LIN {X 0,Y 587.34,Z 320.947,A -85,B 0,C 180,E1 -1290.509,E2 -1290.509} C_VEL
LIN {X 0,Y 587.338,Z 320.944,A -85,B 0,C 180,E1 -1293.397,E2 -1293.397} C_VEL
LIN {X 0,Y 587.293,Z 320.958,A -85,B 0,C 180,E1 -1295.9,E2 -1295.9} C_VEL
LIN {X 0,Y 587.322,Z 320.947,A -85,B 0,C 180,E1 -1298.48,E2 -1298.48} C_VEL
LIN {X 0,Y 587.337,Z 320.944,A -85,B 0,C 180,E1 -1301.157,E2 -1301.157} C_VEL
LIN {X 0,Y 587.317,Z 320.95,A -85,B 0,C 180,E1 -1304.112,E2 -1304.112} C_VEL
LIN {X 0,Y 587.309,Z 320.948,A -85,B 0,C 180,E1 -1306.992,E2 -1306.992} C_VEL
LIN {X 0,Y 587.306,Z 320.955,A -85,B 0,C 180,E1 -1309.744,E2 -1309.744} C_VEL
LIN {X 0,Y 587.312,Z 320.947,A -85,B 0,C 180,E1 -1312.389,E2 -1312.389} C_VEL
LIN {X 0,Y 587.334,Z 320.95,A -85,B 0,C 180,E1 -1315.655,E2 -1315.655} C_VEL
LIN {X 0,Y 587.319,Z 320.946,A -85,B 0,C 180,E1 -1318.229,E2 -1318.229} C_VEL
LIN {X 0,Y 587.324,Z 320.949,A -85,B 0,C 180,E1 -1320.872,E2 -1320.872} C_VEL
LIN {X 0,Y 587.288,Z 320.952,A -85,B 0,C 180,E1 -1323.834,E2 -1323.834} C_VEL
LIN {X 0,Y 587.291,Z 320.955,A -85,B 0,C 180,E1 -1326.739,E2 -1326.739} C_VEL
LIN {X 0,Y 587.343,Z 321.135,A -85,B 0,C 180,E1 -1327.81,E2 -1327.81} C_VEL
LIN {X 0,Y 587.764,Z 325.25,A -85,B 0,C 180,E1 -1328.424,E2 -1328.424} C_VEL
LIN {X 0,Y 587.644,Z 343.161,A -85,B 0,C 180,E1 -1330.991,E2 -1330.991} C_VEL
LIN {X 0,Y 587.518,Z 362.321,A -85,B 0,C 180,E1 -1333.695,E2 -1333.695} C_VEL
LIN {X 0,Y 588.214,Z 367.298,A -85,B 0,C 180,E1 -1333.782,E2 -1333.782} C_VEL
LIN {X 0,Y 588.018,Z 498.318,A -85,B 0,C 180,E1 -1335.419,E2 -1335.419} C_VEL
LIN {X 0,Y 587.927,Z 511.656,A -85,B 0,C 180,E1 -1335.699,E2 -1335.699} C_VEL
LIN {X 0,Y 587.83,Z 526.543,A -85,B 0,C 180,E1 -1336.165,E2 -1336.165} C_VEL
LIN {X 0,Y 587.754,Z 538.919,A -85,B 0,C 180,E1 -1336.691,E2 -1336.691} C_VEL
LIN {X 0,Y 587.657,Z 550.452,A -85,B 0,C 180,E1 -1337.305,E2 -1337.305} C_VEL
LIN {X 0,Y 587.573,Z 561.267,A -85,B 0,C 180,E1 -1338.004,E2 -1338.004} C_VEL
LIN {X 0,Y 587.472,Z 571.624,A -85,B 0,C 180,E1 -1338.807,E2 -1338.807} C_VEL
LIN {X 0,Y 587.377,Z 582.66,A -85,B 0,C 180,E1 -1339.834,E2 -1339.834} C_VEL
LIN {X 0,Y 587.34,Z 591.831,A -85,B 0,C 180,E1 -1340.876,E2 -1340.876} C_VEL
LIN {X 0,Y 587.27,Z 599.476,A -85,B 0,C 180,E1 -1341.916,E2 -1341.916} C_VEL
LIN {X 0,Y 587.211,Z 606.804,A -85,B 0,C 180,E1 -1343.125,E2 -1343.125} C_VEL
LIN {X 0,Y 587.227,Z 611.901,A -85,B 0,C 180,E1 -1344.16,E2 -1344.16} C_VEL
LIN {X 0,Y 587.186,Z 617.246,A -85,B 0,C 180,E1 -1345.537,E2 -1345.537} C_VEL
LIN {X 0,Y 587.182,Z 620.2,A -85,B 0,C 180,E1 -1346.568,E2 -1346.568} C_VEL
LIN {X 0,Y 587.14,Z 622.935,A -85,B 0,C 180,E1 -1347.941,E2 -1347.941} C_VEL
LIN {X 0,Y 587.135,Z 624.296,A -85,B 0,C 180,E1 -1349.313,E2 -1349.313} C_VEL
LIN {X 0,Y 587.136,Z 624.332,A -85,B 0,C 180,E1 -1350.685,E2 -1350.685} C_VEL
LIN {X 0,Y 587.139,Z 623.075,A -85,B 0,C 180,E1 -1352.057,E2 -1352.057} C_VEL
LIN {X 0,Y 587.182,Z 620.438,A -85,B 0,C 180,E1 -1353.43,E2 -1353.43} C_VEL
LIN {X 0,Y 587.14,Z 616.353,A -85,B 0,C 180,E1 -1354.805,E2 -1354.805} C_VEL
LIN {X 0,Y 587.227,Z 612.32,A -85,B 0,C 180,E1 -1355.838,E2 -1355.838} C_VEL
LIN {X 0,Y 587.209,Z 607.297,A -85,B 0,C 180,E1 -1356.873,E2 -1356.873} C_VEL
LIN {X 0,Y 587.268,Z 600.077,A -85,B 0,C 180,E1 -1358.082,E2 -1358.082} C_VEL
LIN {X 0,Y 587.316,Z 591.193,A -85,B 0,C 180,E1 -1359.295,E2 -1359.295} C_VEL
LIN {X 0,Y 587.371,Z 581.851,A -85,B 0,C 180,E1 -1360.338,E2 -1360.338} C_VEL
LIN {X 0,Y 587.478,Z 571.473,A -85,B 0,C 180,E1 -1361.295,E2 -1361.295} C_VEL
LIN {X 0,Y 587.569,Z 560.094,A -85,B 0,C 180,E1 -1362.169,E2 -1362.169} C_VEL
LIN {X 0,Y 587.668,Z 547.487,A -85,B 0,C 180,E1 -1362.957,E2 -1362.957} C_VEL
LIN {X 0,Y 587.8,Z 533.209,A -85,B 0,C 180,E1 -1363.658,E2 -1363.658} C_VEL
LIN {X 0,Y 587.904,Z 520.175,A -85,B 0,C 180,E1 -1364.143,E2 -1364.143} C_VEL
LIN {X 0,Y 587.967,Z 507.624,A -85,B 0,C 180,E1 -1364.488,E2 -1364.488} C_VEL
LIN {X 0,Y 587.997,Z 492.746,A -85,B 0,C 180,E1 -1364.757,E2 -1364.757} C_VEL
LIN {X 0,Y 588.094,Z 365.573,A -85,B 0,C 180,E1 -1366.333,E2 -1366.333} C_VEL
LIN {X 0,Y 587.507,Z 362.182,A -85,B 0,C 180,E1 -1366.415,E2 -1366.415} C_VEL
LIN {X 0,Y 587.674,Z 342.923,A -85,B 0,C 180,E1 -1369.132,E2 -1369.132} C_VEL
LIN {X 0,Y 587.776,Z 324.634,A -85,B 0,C 180,E1 -1371.755,E2 -1371.755} C_VEL
LIN {X 0,Y 587.29,Z 320.956,A -85,B 0,C 180,E1 -1372.329,E2 -1372.329} C_VEL
LIN {X 0,Y 587.291,Z 320.956,A -85,B 0,C 180,E1 -1374.76,E2 -1374.76} C_VEL
LIN {X 0,Y 587.291,Z 320.95,A -85,B 0,C 180,E1 -1377.681,E2 -1377.681} C_VEL
LIN {X 0,Y 587.286,Z 320.95,A -85,B 0,C 180,E1 -1380.171,E2 -1380.171} C_VEL
LIN {X 0,Y 587.32,Z 320.95,A -85,B 0,C 180,E1 -1382.579,E2 -1382.579} C_VEL
LIN {X 0,Y 587.316,Z 320.954,A -85,B 0,C 180,E1 -1385.055,E2 -1385.055} C_VEL
LIN {X 0,Y 587.302,Z 320.947,A -85,B 0,C 180,E1 -1387.833,E2 -1387.833} C_VEL
LIN {X 0,Y 587.29,Z 320.95,A -85,B 0,C 180,E1 -1390.254,E2 -1390.254} C_VEL
LIN {X 0,Y 587.281,Z 320.956,A -85,B 0,C 180,E1 -1393.114,E2 -1393.114} C_VEL
LIN {X 0,Y 587.301,Z 320.948,A -85,B 0,C 180,E1 -1396.047,E2 -1396.047} C_VEL
LIN {X 0,Y 587.318,Z 320.955,A -85,B 0,C 180,E1 -1398.925,E2 -1398.925} C_VEL
LIN {X 0,Y 587.291,Z 320.948,A -85,B 0,C 180,E1 -1401.517,E2 -1401.517} C_VEL
LIN {X 0,Y 587.262,Z 320.953,A -85,B 0,C 180,E1 -1404.098,E2 -1404.098} C_VEL
LIN {X 0,Y 587.319,Z 320.953,A -85,B 0,C 180,E1 -1406.888,E2 -1406.888} C_VEL
LIN {X 0,Y 587.293,Z 320.949,A -85,B 0,C 180,E1 -1409.494,E2 -1409.494} C_VEL
LIN {X 0,Y 587.275,Z 320.952,A -85,B 0,C 180,E1 -1411.4,E2 -1411.4} C_VEL
LIN {X 0,Y 587.289,Z 320.947,A -85,B 0,C 180,E1 -1413.829,E2 -1413.829} C_VEL
LIN {X 0,Y 587.284,Z 320.96,A -85,B 0,C 180,E1 -1416.74,E2 -1416.74} C_VEL
LIN {X 0,Y 587.29,Z 320.947,A -85,B 0,C 180,E1 -1419.694,E2 -1419.694} C_VEL
LIN {X 0,Y 587.265,Z 320.951,A -85,B 0,C 180,E1 -1421.871,E2 -1421.871} C_VEL
LIN {X 0,Y 587.279,Z 320.951,A -85,B 0,C 180,E1 -1424.023,E2 -1424.023} C_VEL
LIN {X 0,Y 587.268,Z 320.958,A -85,B 0,C 180,E1 -1426.857,E2 -1426.857} C_VEL
LIN {X 0,Y 587.321,Z 320.95,A -85,B 0,C 180,E1 -1428.962,E2 -1428.962} C_VEL
LIN {X 0,Y 587.297,Z 320.948,A -85,B 0,C 180,E1 -1431.744,E2 -1431.744} C_VEL
LIN {X 0,Y 587.333,Z 320.952,A -85,B 0,C 180,E1 -1434.507,E2 -1434.507} C_VEL
LIN {X 0,Y 587.327,Z 320.945,A -85,B 0,C 180,E1 -1437.256,E2 -1437.256} C_VEL
LIN {X 0,Y 587.342,Z 320.944,A -85,B 0,C 180,E1 -1440,E2 -1440} C_VEL
LIN {X 0,Y 587.356,Z 320.947,A -85,B 0,C 180,E1 -1442.743,E2 -1442.743} C_VEL
LIN {X 0,Y 587.304,Z 320.947,A -85,B 0,C 180,E1 -1445.493,E2 -1445.493} C_VEL
LIN {X 0,Y 587.284,Z 320.949,A -85,B 0,C 180,E1 -1447.564,E2 -1447.564} C_VEL
LIN {X 0,Y 587.284,Z 320.957,A -85,B 0,C 180,E1 -1450.341,E2 -1450.341} C_VEL
LIN {X 0,Y 587.277,Z 320.951,A -85,B 0,C 180,E1 -1453.143,E2 -1453.143} C_VEL
LIN {X 0,Y 587.297,Z 320.948,A -85,B 0,C 180,E1 -1455.264,E2 -1455.264} C_VEL
LIN {X 0,Y 587.266,Z 320.951,A -85,B 0,C 180,E1 -1457.409,E2 -1457.409} C_VEL
LIN {X 0,Y 587.283,Z 320.95,A -85,B 0,C 180,E1 -1459.577,E2 -1459.577} C_VEL
LIN {X 0,Y 587.292,Z 320.949,A -85,B 0,C 180,E1 -1461.775,E2 -1461.775} C_VEL
LIN {X 0,Y 587.289,Z 320.953,A -85,B 0,C 180,E1 -1464.761,E2 -1464.761} C_VEL
LIN {X 0,Y 587.285,Z 320.95,A -85,B 0,C 180,E1 -1467.684,E2 -1467.684} C_VEL
LIN {X 0,Y 587.294,Z 320.954,A -85,B 0,C 180,E1 -1470.172,E2 -1470.172} C_VEL
LIN {X 0,Y 587.314,Z 320.946,A -85,B 0,C 180,E1 -1473.111,E2 -1473.111} C_VEL
LIN {X 0,Y 587.259,Z 320.956,A -85,B 0,C 180,E1 -1475.902,E2 -1475.902} C_VEL
LIN {X 0,Y 587.295,Z 320.955,A -85,B 0,C 180,E1 -1478.482,E2 -1478.482} C_VEL
LIN {X 0,Y 587.272,Z 320.951,A -85,B 0,C 180,E1 -1481.162,E2 -1481.162} C_VEL
LIN {X 0,Y 587.29,Z 320.957,A -85,B 0,C 180,E1 -1484.112,E2 -1484.112} C_VEL
LIN {X 0,Y 587.259,Z 320.953,A -85,B 0,C 180,E1 -1486.991,E2 -1486.991} C_VEL
LIN {X 0,Y 587.28,Z 320.957,A -85,B 0,C 180,E1 -1489.986,E2 -1489.986} C_VEL
LIN {X 0,Y 587.299,Z 320.955,A -85,B 0,C 180,E1 -1492.391,E2 -1492.391} C_VEL
LIN {X 0,Y 587.312,Z 320.949,A -85,B 0,C 180,E1 -1495.658,E2 -1495.658} C_VEL
LIN {X 0,Y 587.324,Z 320.954,A -85,B 0,C 180,E1 -1498.232,E2 -1498.232} C_VEL
LIN {X 0,Y 587.29,Z 320.949,A -85,B 0,C 180,E1 -1500.877,E2 -1500.877} C_VEL
LIN {X 0,Y 587.295,Z 320.954,A -85,B 0,C 180,E1 -1503.832,E2 -1503.832} C_VEL
LIN {X 0,Y 587.316,Z 321.138,A -85,B 0,C 180,E1 -1506.742,E2 -1506.742} C_VEL
LIN {X 0,Y 587.851,Z 325.282,A -85,B 0,C 180,E1 -1507.339,E2 -1507.339} C_VEL
LIN {X 0,Y 587.746,Z 345.308,A -85,B 0,C 180,E1 -1510.076,E2 -1510.076} C_VEL
LIN {X 0,Y 587.586,Z 367.907,A -85,B 0,C 180,E1 -1513.11,E2 -1513.11} C_VEL
LIN {X 0,Y 587.592,Z 372.251,A -85,B 0,C 180,E1 -1513.656,E2 -1513.656} C_VEL
LIN {X 0,Y 588.201,Z 376.337,A -85,B 0,C 180,E1 -1513.724,E2 -1513.724} C_VEL
LIN {X 0,Y 587.986,Z 509.948,A -85,B 0,C 180,E1 -1515.398,E2 -1515.398} C_VEL
LIN {X 0,Y 587.945,Z 524.277,A -85,B 0,C 180,E1 -1515.724,E2 -1515.724} C_VEL
LIN {X 0,Y 587.824,Z 537.74,A -85,B 0,C 180,E1 -1516.167,E2 -1516.167} C_VEL
LIN {X 0,Y 587.726,Z 551.664,A -85,B 0,C 180,E1 -1516.781,E2 -1516.781} C_VEL
LIN {X 0,Y 587.626,Z 564.117,A -85,B 0,C 180,E1 -1517.482,E2 -1517.482} C_VEL
LIN {X 0,Y 587.512,Z 576.654,A -85,B 0,C 180,E1 -1518.355,E2 -1518.355} C_VEL
LIN {X 0,Y 587.444,Z 587.848,A -85,B 0,C 180,E1 -1519.315,E2 -1519.315} C_VEL
LIN {X 0,Y 587.319,Z 597.86,A -85,B 0,C 180,E1 -1520.357,E2 -1520.357} C_VEL
LIN {X 0,Y 587.277,Z 606.179,A -85,B 0,C 180,E1 -1521.398,E2 -1521.398} C_VEL
LIN {X 0,Y 587.243,Z 614.133,A -85,B 0,C 180,E1 -1522.609,E2 -1522.609} C_VEL
LIN {X 0,Y 587.202,Z 620.532,A -85,B 0,C 180,E1 -1523.817,E2 -1523.817} C_VEL
LIN {X 0,Y 587.16,Z 624.965,A -85,B 0,C 180,E1 -1524.851,E2 -1524.851} C_VEL
LIN {X 0,Y 587.179,Z 628.447,A -85,B 0,C 180,E1 -1525.883,E2 -1525.883} C_VEL
LIN {X 0,Y 587.13,Z 631.835,A -85,B 0,C 180,E1 -1527.257,E2 -1527.257} C_VEL
LIN {X 0,Y 587.141,Z 633.833,A -85,B 0,C 180,E1 -1528.629,E2 -1528.629} C_VEL
LIN {X 0,Y 587.135,Z 634.5,A -85,B 0,C 180,E1 -1530.001,E2 -1530.001} C_VEL
LIN {X 0,Y 587.141,Z 633.831,A -85,B 0,C 180,E1 -1531.373,E2 -1531.373} C_VEL
LIN {X 0,Y 587.13,Z 631.829,A -85,B 0,C 180,E1 -1532.745,E2 -1532.745} C_VEL
LIN {X 0,Y 587.179,Z 628.439,A -85,B 0,C 180,E1 -1534.119,E2 -1534.119} C_VEL
LIN {X 0,Y 587.199,Z 623.564,A -85,B 0,C 180,E1 -1535.495,E2 -1535.495} C_VEL
LIN {X 0,Y 587.21,Z 617.047,A -85,B 0,C 180,E1 -1536.875,E2 -1536.875} C_VEL
LIN {X 0,Y 587.269,Z 609.793,A -85,B 0,C 180,E1 -1538.084,E2 -1538.084} C_VEL
LIN {X 0,Y 587.322,Z 600.815,A -85,B 0,C 180,E1 -1539.297,E2 -1539.297} C_VEL
LIN {X 0,Y 587.372,Z 591.382,A -85,B 0,C 180,E1 -1540.34,E2 -1540.34} C_VEL
LIN {X 0,Y 587.476,Z 581.019,A -85,B 0,C 180,E1 -1541.291,E2 -1541.291} C_VEL
LIN {X 0,Y 587.576,Z 569.417,A -85,B 0,C 180,E1 -1542.171,E2 -1542.171} C_VEL
LIN {X 0,Y 587.673,Z 556.63,A -85,B 0,C 180,E1 -1542.959,E2 -1542.959} C_VEL
LIN {X 0,Y 587.795,Z 544.14,A -85,B 0,C 180,E1 -1543.572,E2 -1543.572} C_VEL
LIN {X 0,Y 587.908,Z 530.693,A -85,B 0,C 180,E1 -1544.082,E2 -1544.082} C_VEL
LIN {X 0,Y 587.946,Z 516.96,A -85,B 0,C 180,E1 -1544.462,E2 -1544.462} C_VEL
LIN {X 0,Y 588.015,Z 502.535,A -85,B 0,C 180,E1 -1544.714,E2 -1544.714} C_VEL
LIN {X 0,Y 588.141,Z 375.219,A -85,B 0,C 180,E1 -1546.291,E2 -1546.291} C_VEL
LIN {X 0,Y 587.563,Z 371.811,A -85,B 0,C 180,E1 -1546.371,E2 -1546.371} C_VEL
LIN {X 0,Y 587.696,Z 351.121,A -85,B 0,C 180,E1 -1549.139,E2 -1549.139} C_VEL
LIN {X 0,Y 587.867,Z 330.521,A -85,B 0,C 180,E1 -1551.938,E2 -1551.938} C_VEL
LIN {X 0,Y 587.608,Z 322.589,A -85,B 0,C 180,E1 -1553.044,E2 -1553.044} C_VEL
LIN {X 0,Y 587.297,Z 320.956,A -85,B 0,C 180,E1 -1553.307,E2 -1553.307} C_VEL
LIN {X 0,Y 587.296,Z 320.952,A -85,B 0,C 180,E1 -1556.281,E2 -1556.281} C_VEL
LIN {X 0,Y 587.302,Z 320.951,A -85,B 0,C 180,E1 -1559.125,E2 -1559.125} C_VEL
LIN {X 0,Y 587.318,Z 320.95,A -85,B 0,C 180,E1 -1561.831,E2 -1561.831} C_VEL
LIN {X 0,Y 587.341,Z 320.943,A -85,B 0,C 180,E1 -1564.347,E2 -1564.347} C_VEL
LIN {X 0,Y 587.346,Z 320.946,A -85,B 0,C 180,E1 -1567.608,E2 -1567.608} C_VEL
LIN {X 0,Y 587.318,Z 320.946,A -85,B 0,C 180,E1 -1570.255,E2 -1570.255} C_VEL
LIN {X 0,Y 587.318,Z 320.953,A -85,B 0,C 180,E1 -1573.118,E2 -1573.118} C_VEL
LIN {X 0,Y 587.328,Z 320.946,A -85,B 0,C 180,E1 -1576.05,E2 -1576.05} C_VEL
LIN {X 0,Y 587.339,Z 320.949,A -85,B 0,C 180,E1 -1578.926,E2 -1578.926} C_VEL
LIN {X 0,Y 587.325,Z 320.945,A -85,B 0,C 180,E1 -1581.52,E2 -1581.52} C_VEL
LIN {X 0,Y 587.299,Z 320.957,A -85,B 0,C 180,E1 -1584.463,E2 -1584.463} C_VEL
LIN {X 0,Y 587.341,Z 320.945,A -85,B 0,C 180,E1 -1586.889,E2 -1586.889} C_VEL
LIN {X 0,Y 587.334,Z 320.949,A -85,B 0,C 180,E1 -1589.83,E2 -1589.83} C_VEL
LIN {X 0,Y 587.304,Z 320.954,A -85,B 0,C 180,E1 -1592.317,E2 -1592.317} C_VEL
LIN {X 0,Y 587.31,Z 320.949,A -85,B 0,C 180,E1 -1595.24,E2 -1595.24} C_VEL
LIN {X 0,Y 587.302,Z 320.954,A -85,B 0,C 180,E1 -1598.225,E2 -1598.225} C_VEL
LIN {X 0,Y 587.312,Z 321.009,A -85,B 0,C 180,E1 -1598.548,E2 -1598.548} C_VEL
LIN {X 0,Y 587.665,Z 325.965,A -85,B 0,C 180,E1 -1599.342,E2 -1599.342} C_VEL
LIN {X 0,Y 587.534,Z 343.467,A -85,B 0,C 180,E1 -1602.06,E2 -1602.06} C_VEL
LIN {X 0,Y 587.449,Z 362.136,A -85,B 0,C 180,E1 -1604.918,E2 -1604.918} C_VEL
LIN {X 0,Y 587.389,Z 372.929,A -85,B 0,C 180,E1 -1606.552,E2 -1606.552} C_VEL
LIN {X 0,Y 587.889,Z 377.929,A -85,B 0,C 180,E1 -1606.63,E2 -1606.63} C_VEL
LIN {X 0,Y 587.74,Z 480.331,A -85,B 0,C 180,E1 -1607.899,E2 -1607.899} C_VEL
LIN {X 0,Y 587.703,Z 493.687,A -85,B 0,C 180,E1 -1608.205,E2 -1608.205} C_VEL
LIN {X 0,Y 587.597,Z 506.208,A -85,B 0,C 180,E1 -1608.633,E2 -1608.633} C_VEL
LIN {X 0,Y 587.583,Z 517.258,A -85,B 0,C 180,E1 -1609.142,E2 -1609.142} C_VEL
LIN {X 0,Y 587.44,Z 527.713,A -85,B 0,C 180,E1 -1609.749,E2 -1609.749} C_VEL
LIN {X 0,Y 587.381,Z 538.488,A -85,B 0,C 180,E1 -1610.531,E2 -1610.531} C_VEL
LIN {X 0,Y 587.323,Z 548.152,A -85,B 0,C 180,E1 -1611.398,E2 -1611.398} C_VEL
LIN {X 0,Y 587.274,Z 556.076,A -85,B 0,C 180,E1 -1612.263,E2 -1612.263} C_VEL
LIN {X 0,Y 587.233,Z 562.636,A -85,B 0,C 180,E1 -1613.126,E2 -1613.126} C_VEL
LIN {X 0,Y 587.237,Z 569.112,A -85,B 0,C 180,E1 -1614.161,E2 -1614.161} C_VEL
LIN {X 0,Y 587.146,Z 574.245,A -85,B 0,C 180,E1 -1615.194,E2 -1615.194} C_VEL
LIN {X 0,Y 587.213,Z 578.247,A -85,B 0,C 180,E1 -1616.226,E2 -1616.226} C_VEL
LIN {X 0,Y 587.132,Z 581.188,A -85,B 0,C 180,E1 -1617.256,E2 -1617.256} C_VEL
LIN {X 0,Y 587.139,Z 582.618,A -85,B 0,C 180,E1 -1617.942,E2 -1617.942} C_VEL
LIN {X 0,Y 587.148,Z 583.634,A -85,B 0,C 180,E1 -1618.628,E2 -1618.628} C_VEL
LIN {X 0,Y 587.137,Z 584.496,A -85,B 0,C 180,E1 -1620,E2 -1620} C_VEL
LIN {X 0,Y 587.14,Z 584.321,A -85,B 0,C 180,E1 -1620.686,E2 -1620.686} C_VEL
LIN {X 0,Y 587.138,Z 582.767,A -85,B 0,C 180,E1 -1622.058,E2 -1622.058} C_VEL
LIN {X 0,Y 587.133,Z 581.398,A -85,B 0,C 180,E1 -1622.744,E2 -1622.744} C_VEL
LIN {X 0,Y 587.213,Z 578.532,A -85,B 0,C 180,E1 -1623.774,E2 -1623.774} C_VEL
LIN {X 0,Y 587.147,Z 574.644,A -85,B 0,C 180,E1 -1624.806,E2 -1624.806} C_VEL
LIN {X 0,Y 587.229,Z 569.592,A -85,B 0,C 180,E1 -1625.839,E2 -1625.839} C_VEL
LIN {X 0,Y 587.231,Z 563.277,A -85,B 0,C 180,E1 -1626.874,E2 -1626.874} C_VEL
LIN {X 0,Y 587.288,Z 555.374,A -85,B 0,C 180,E1 -1627.91,E2 -1627.91} C_VEL
LIN {X 0,Y 587.325,Z 547.296,A -85,B 0,C 180,E1 -1628.776,E2 -1628.776} C_VEL
LIN {X 0,Y 587.386,Z 537.461,A -85,B 0,C 180,E1 -1629.643,E2 -1629.643} C_VEL
LIN {X 0,Y 587.484,Z 526.401,A -85,B 0,C 180,E1 -1630.425,E2 -1630.425} C_VEL
LIN {X 0,Y 587.566,Z 514.121,A -85,B 0,C 180,E1 -1631.106,E2 -1631.106} C_VEL
LIN {X 0,Y 587.625,Z 502.329,A -85,B 0,C 180,E1 -1631.607,E2 -1631.607} C_VEL
LIN {X 0,Y 587.713,Z 489.755,A -85,B 0,C 180,E1 -1631.992,E2 -1631.992} C_VEL
LIN {X 0,Y 587.757,Z 476.243,A -85,B 0,C 180,E1 -1632.254,E2 -1632.254} C_VEL
LIN {X 0,Y 587.779,Z 461.163,A -85,B 0,C 180,E1 -1632.441,E2 -1632.441} C_VEL
LIN {X 0,Y 587.15,Z 455.354,A -85,B 0,C 180,E1 -1632.526,E2 -1632.526} C_VEL
LIN {X 0,Y 581.565,Z 436.661,A -85,B 0,C 180,E1 -1632.879,E2 -1632.879} C_VEL
LIN {X 0,Y 580.932,Z 430.852,A -85,B 0,C 180,E1 -1632.966,E2 -1632.966} C_VEL
LIN {X 0,Y 580.87,Z 376.245,A -85,B 0,C 180,E1 -1633.647,E2 -1633.647} C_VEL
LIN {X 0,Y 580.384,Z 372.937,A -85,B 0,C 180,E1 -1633.703,E2 -1633.703} C_VEL
LIN {X 0,Y 580.491,Z 354.552,A -85,B 0,C 180,E1 -1636.53,E2 -1636.53} C_VEL
LIN {X 0,Y 580.64,Z 335.922,A -85,B 0,C 180,E1 -1639.435,E2 -1639.435} C_VEL
LIN {X 0,Y 580.682,Z 324.199,A -85,B 0,C 180,E1 -1641.29,E2 -1641.29} C_VEL
LIN {X 0,Y 580.329,Z 321.823,A -85,B 0,C 180,E1 -1641.723,E2 -1641.723} C_VEL
LIN {X 0,Y 580.326,Z 321.82,A -85,B 0,C 180,E1 -1644.73,E2 -1644.73} C_VEL
LIN {X 0,Y 580.286,Z 321.822,A -85,B 0,C 180,E1 -1647.402,E2 -1647.402} C_VEL
LIN {X 0,Y 580.29,Z 321.825,A -85,B 0,C 180,E1 -1649.773,E2 -1649.773} C_VEL
LIN {X 0,Y 580.3,Z 321.828,A -85,B 0,C 180,E1 -1652.201,E2 -1652.201} C_VEL
LIN {X 0,Y 580.29,Z 321.822,A -85,B 0,C 180,E1 -1654.696,E2 -1654.696} C_VEL
LIN {X 0,Y 580.292,Z 321.822,A -85,B 0,C 180,E1 -1657.269,E2 -1657.269} C_VEL
LIN {X 0,Y 580.291,Z 321.824,A -85,B 0,C 180,E1 -1660.27,E2 -1660.27} C_VEL
LIN {X 0,Y 580.263,Z 321.825,A -85,B 0,C 180,E1 -1662.708,E2 -1662.708} C_VEL
LIN {X 0,Y 580.255,Z 321.834,A -85,B 0,C 180,E1 -1665.611,E2 -1665.611} C_VEL
LIN {X 0,Y 580.255,Z 321.827,A -85,B 0,C 180,E1 -1668.228,E2 -1668.228} C_VEL
LIN {X 0,Y 580.267,Z 321.826,A -85,B 0,C 180,E1 -1670.963,E2 -1670.963} C_VEL
LIN {X 0,Y 580.247,Z 321.835,A -85,B 0,C 180,E1 -1673.594,E2 -1673.594} C_VEL
LIN {X 0,Y 580.268,Z 321.825,A -85,B 0,C 180,E1 -1676.141,E2 -1676.141} C_VEL
LIN {X 0,Y 580.254,Z 321.827,A -85,B 0,C 180,E1 -1678.612,E2 -1678.612} C_VEL
LIN {X 0,Y 580.269,Z 321.83,A -85,B 0,C 180,E1 -1681.022,E2 -1681.022} C_VEL
LIN {X 0,Y 580.242,Z 321.831,A -85,B 0,C 180,E1 -1683.676,E2 -1683.676} C_VEL
LIN {X 0,Y 580.241,Z 321.831,A -85,B 0,C 180,E1 -1686.44,E2 -1686.44} C_VEL
LIN {X 0,Y 580.296,Z 321.935,A -85,B 0,C 180,E1 -1687.643,E2 -1687.643} C_VEL
LIN {X 0,Y 580.845,Z 326.548,A -85,B 0,C 180,E1 -1688.343,E2 -1688.343} C_VEL
LIN {X 0,Y 580.696,Z 344.355,A -85,B 0,C 180,E1 -1690.926,E2 -1690.926} C_VEL
LIN {X 0,Y 580.528,Z 362.325,A -85,B 0,C 180,E1 -1693.493,E2 -1693.493} C_VEL
LIN {X 0,Y 581.395,Z 367.344,A -85,B 0,C 180,E1 -1693.586,E2 -1693.586} C_VEL
LIN {X 0,Y 581.137,Z 498.296,A -85,B 0,C 180,E1 -1695.242,E2 -1695.242} C_VEL
LIN {X 0,Y 581.031,Z 511.361,A -85,B 0,C 180,E1 -1695.518,E2 -1695.518} C_VEL
LIN {X 0,Y 580.985,Z 524.976,A -85,B 0,C 180,E1 -1695.939,E2 -1695.939} C_VEL
LIN {X 0,Y 580.824,Z 538.917,A -85,B 0,C 180,E1 -1696.53,E2 -1696.53} C_VEL
LIN {X 0,Y 580.702,Z 550.445,A -85,B 0,C 180,E1 -1697.15,E2 -1697.15} C_VEL
LIN {X 0,Y 580.597,Z 561.261,A -85,B 0,C 180,E1 -1697.858,E2 -1697.858} C_VEL
LIN {X 0,Y 580.46,Z 572.357,A -85,B 0,C 180,E1 -1698.732,E2 -1698.732} C_VEL
LIN {X 0,Y 580.348,Z 582.666,A -85,B 0,C 180,E1 -1699.71,E2 -1699.71} C_VEL
LIN {X 0,Y 580.296,Z 591.834,A -85,B 0,C 180,E1 -1700.765,E2 -1700.765} C_VEL
LIN {X 0,Y 580.194,Z 599.472,A -85,B 0,C 180,E1 -1701.816,E2 -1701.816} C_VEL
LIN {X 0,Y 580.149,Z 604.882,A -85,B 0,C 180,E1 -1702.691,E2 -1702.691} C_VEL
LIN {X 0,Y 580.104,Z 610.309,A -85,B 0,C 180,E1 -1703.739,E2 -1703.739} C_VEL
LIN {X 0,Y 580.077,Z 614.768,A -85,B 0,C 180,E1 -1704.786,E2 -1704.786} C_VEL
LIN {X 0,Y 580.104,Z 618.311,A -85,B 0,C 180,E1 -1705.83,E2 -1705.83} C_VEL
LIN {X 0,Y 580.041,Z 621.721,A -85,B 0,C 180,E1 -1707.221,E2 -1707.221} C_VEL
LIN {X 0,Y 580.045,Z 623.764,A -85,B 0,C 180,E1 -1708.61,E2 -1708.61} C_VEL
LIN {X 0,Y 580.037,Z 624.496,A -85,B 0,C 180,E1 -1709.999,E2 -1709.999} C_VEL
LIN {X 0,Y 580.042,Z 623.867,A -85,B 0,C 180,E1 -1711.388,E2 -1711.388} C_VEL
LIN {X 0,Y 580.039,Z 621.901,A -85,B 0,C 180,E1 -1712.777,E2 -1712.777} C_VEL
LIN {X 0,Y 580.108,Z 620.437,A -85,B 0,C 180,E1 -1713.472,E2 -1713.472} C_VEL
LIN {X 0,Y 580.046,Z 616.347,A -85,B 0,C 180,E1 -1714.864,E2 -1714.864} C_VEL
LIN {X 0,Y 580.133,Z 612.309,A -85,B 0,C 180,E1 -1715.909,E2 -1715.909} C_VEL
LIN {X 0,Y 580.141,Z 607.295,A -85,B 0,C 180,E1 -1716.957,E2 -1716.957} C_VEL
LIN {X 0,Y 580.192,Z 600.066,A -85,B 0,C 180,E1 -1718.182,E2 -1718.182} C_VEL
LIN {X 0,Y 580.284,Z 592.546,A -85,B 0,C 180,E1 -1719.233,E2 -1719.233} C_VEL
LIN {X 0,Y 580.346,Z 583.517,A -85,B 0,C 180,E1 -1720.288,E2 -1720.288} C_VEL
LIN {X 0,Y 580.492,Z 572.513,A -85,B 0,C 180,E1 -1721.345,E2 -1721.345} C_VEL
LIN {X 0,Y 580.575,Z 561.309,A -85,B 0,C 180,E1 -1722.229,E2 -1722.229} C_VEL
LIN {X 0,Y 580.683,Z 550.497,A -85,B 0,C 180,E1 -1722.937,E2 -1722.937} C_VEL
LIN {X 0,Y 580.861,Z 537.18,A -85,B 0,C 180,E1 -1723.646,E2 -1723.646} C_VEL
LIN {X 0,Y 580.992,Z 524.262,A -85,B 0,C 180,E1 -1724.175,E2 -1724.175} C_VEL
LIN {X 0,Y 581.055,Z 510.601,A -85,B 0,C 180,E1 -1724.59,E2 -1724.59} C_VEL
LIN {X 0,Y 581.121,Z 498.452,A -85,B 0,C 180,E1 -1724.846,E2 -1724.846} C_VEL
LIN {X 0,Y 581.312,Z 366.587,A -85,B 0,C 180,E1 -1726.516,E2 -1726.516} C_VEL
LIN {X 0,Y 580.522,Z 362.178,A -85,B 0,C 180,E1 -1726.618,E2 -1726.618} C_VEL
LIN {X 0,Y 580.751,Z 342.169,A -85,B 0,C 180,E1 -1729.478,E2 -1729.478} C_VEL
LIN {X 0,Y 580.86,Z 326.03,A -85,B 0,C 180,E1 -1731.822,E2 -1731.822} C_VEL
LIN {X 0,Y 580.254,Z 321.833,A -85,B 0,C 180,E1 -1732.474,E2 -1732.474} C_VEL
LIN {X 0,Y 580.267,Z 321.834,A -85,B 0,C 180,E1 -1735.08,E2 -1735.08} C_VEL
LIN {X 0,Y 580.238,Z 321.828,A -85,B 0,C 180,E1 -1737.847,E2 -1737.847} C_VEL
LIN {X 0,Y 580.25,Z 321.832,A -85,B 0,C 180,E1 -1740.688,E2 -1740.688} C_VEL
LIN {X 0,Y 580.269,Z 321.829,A -85,B 0,C 180,E1 -1743.311,E2 -1743.311} C_VEL
LIN {X 0,Y 580.232,Z 321.829,A -85,B 0,C 180,E1 -1745.754,E2 -1745.754} C_VEL
LIN {X 0,Y 580.267,Z 321.824,A -85,B 0,C 180,E1 -1748.146,E2 -1748.146} C_VEL
LIN {X 0,Y 580.269,Z 321.833,A -85,B 0,C 180,E1 -1750.844,E2 -1750.844} C_VEL
LIN {X 0,Y 580.225,Z 321.829,A -85,B 0,C 180,E1 -1753.661,E2 -1753.661} C_VEL
LIN {X 0,Y 580.254,Z 321.831,A -85,B 0,C 180,E1 -1756.61,E2 -1756.61} C_VEL
LIN {X 0,Y 580.263,Z 321.824,A -85,B 0,C 180,E1 -1759.731,E2 -1759.731} C_VEL
LIN {X 0,Y 580.271,Z 321.831,A -85,B 0,C 180,E1 -1762.729,E2 -1762.729} C_VEL
LIN {X 0,Y 580.269,Z 321.824,A -85,B 0,C 180,E1 -1765.443,E2 -1765.443} C_VEL
LIN {X 0,Y 580.27,Z 321.822,A -85,B 0,C 180,E1 -1767.971,E2 -1767.971} C_VEL
LIN {X 0,Y 580.262,Z 321.83,A -85,B 0,C 180,E1 -1771.022,E2 -1771.022} C_VEL
LIN {X 0,Y 580.246,Z 321.824,A -85,B 0,C 180,E1 -1773.672,E2 -1773.672} C_VEL
LIN {X 0,Y 580.234,Z 321.833,A -85,B 0,C 180,E1 -1776.44,E2 -1776.44} C_VEL
LIN {X 0,Y 580.244,Z 321.826,A -85,B 0,C 180,E1 -1779.436,E2 -1779.436} C_VEL
LIN {X 0,Y 580.224,Z 321.827,A -85,B 0,C 180,E1 -1781.644,E2 -1781.644} C_VEL
LIN {X 0,Y 580.23,Z 321.828,A -85,B 0,C 180,E1 -1783.824,E2 -1783.824} C_VEL
LIN {X 0,Y 580.266,Z 321.825,A -85,B 0,C 180,E1 -1785.981,E2 -1785.981} C_VEL
LIN {X 0,Y 580.29,Z 321.828,A -85,B 0,C 180,E1 -1788.827,E2 -1788.827} C_VEL
LIN {X 0,Y 580.271,Z 321.823,A -85,B 0,C 180,E1 -1791.643,E2 -1791.643} C_VEL
LIN {X 0,Y 580.296,Z 321.828,A -85,B 0,C 180,E1 -1794.44,E2 -1794.44} C_VEL
LIN {X 0,Y 580.297,Z 321.821,A -85,B 0,C 180,E1 -1797.223,E2 -1797.223} C_VEL
LIN {X 0,Y 580.312,Z 321.819,A -85,B 0,C 180,E1 -1800,E2 -1800} C_VEL
LIN {X 0,Y 580.318,Z 321.823,A -85,B 0,C 180,E1 -1802.777,E2 -1802.777} C_VEL
LIN {X 0,Y 580.273,Z 321.823,A -85,B 0,C 180,E1 -1805.56,E2 -1805.56} C_VEL
LIN {X 0,Y 580.237,Z 321.827,A -85,B 0,C 180,E1 -1807.657,E2 -1807.657} C_VEL
LIN {X 0,Y 580.248,Z 321.836,A -85,B 0,C 180,E1 -1810.468,E2 -1810.468} C_VEL
LIN {X 0,Y 580.273,Z 321.831,A -85,B 0,C 180,E1 -1812.592,E2 -1812.592} C_VEL
LIN {X 0,Y 580.264,Z 321.829,A -85,B 0,C 180,E1 -1814.735,E2 -1814.735} C_VEL
LIN {X 0,Y 580.232,Z 321.828,A -85,B 0,C 180,E1 -1817.626,E2 -1817.626} C_VEL
LIN {X 0,Y 580.261,Z 321.826,A -85,B 0,C 180,E1 -1819.824,E2 -1819.824} C_VEL
LIN {X 0,Y 580.244,Z 321.829,A -85,B 0,C 180,E1 -1822.054,E2 -1822.054} C_VEL
LIN {X 0,Y 580.248,Z 321.831,A -85,B 0,C 180,E1 -1824.718,E2 -1824.718} C_VEL
LIN {X 0,Y 580.228,Z 321.828,A -85,B 0,C 180,E1 -1827.405,E2 -1827.405} C_VEL
LIN {X 0,Y 580.246,Z 321.826,A -85,B 0,C 180,E1 -1829.775,E2 -1829.775} C_VEL
LIN {X 0,Y 580.272,Z 321.831,A -85,B 0,C 180,E1 -1832.202,E2 -1832.202} C_VEL
LIN {X 0,Y 580.256,Z 321.829,A -85,B 0,C 180,E1 -1834.699,E2 -1834.699} C_VEL
LIN {X 0,Y 580.251,Z 321.826,A -85,B 0,C 180,E1 -1837.272,E2 -1837.272} C_VEL
LIN {X 0,Y 580.255,Z 321.836,A -85,B 0,C 180,E1 -1840.269,E2 -1840.269} C_VEL
LIN {X 0,Y 580.242,Z 321.83,A -85,B 0,C 180,E1 -1842.71,E2 -1842.71} C_VEL
LIN {X 0,Y 580.224,Z 321.831,A -85,B 0,C 180,E1 -1845.614,E2 -1845.614} C_VEL
LIN {X 0,Y 580.223,Z 321.84,A -85,B 0,C 180,E1 -1848.228,E2 -1848.228} C_VEL
LIN {X 0,Y 580.229,Z 321.829,A -85,B 0,C 180,E1 -1850.963,E2 -1850.963} C_VEL
LIN {X 0,Y 580.222,Z 321.831,A -85,B 0,C 180,E1 -1853.595,E2 -1853.595} C_VEL
LIN {X 0,Y 580.255,Z 321.835,A -85,B 0,C 180,E1 -1856.143,E2 -1856.143} C_VEL
LIN {X 0,Y 580.255,Z 321.828,A -85,B 0,C 180,E1 -1858.615,E2 -1858.615} C_VEL
LIN {X 0,Y 580.234,Z 321.828,A -85,B 0,C 180,E1 -1861.022,E2 -1861.022} C_VEL
LIN {X 0,Y 580.246,Z 321.831,A -85,B 0,C 180,E1 -1863.675,E2 -1863.675} C_VEL
LIN {X 0,Y 580.275,Z 321.877,A -85,B 0,C 180,E1 -1866.547,E2 -1866.547} C_VEL
LIN {X 0,Y 580.954,Z 326.509,A -85,B 0,C 180,E1 -1867.226,E2 -1867.226} C_VEL
LIN {X 0,Y 580.82,Z 345.308,A -85,B 0,C 180,E1 -1869.829,E2 -1869.829} C_VEL
LIN {X 0,Y 580.635,Z 367.06,A -85,B 0,C 180,E1 -1872.787,E2 -1872.787} C_VEL
LIN {X 0,Y 580.568,Z 371.911,A -85,B 0,C 180,E1 -1873.44,E2 -1873.44} C_VEL
LIN {X 0,Y 581.396,Z 377.505,A -85,B 0,C 180,E1 -1873.543,E2 -1873.543} C_VEL
LIN {X 0,Y 581.135,Z 509.947,A -85,B 0,C 180,E1 -1875.222,E2 -1875.222} C_VEL
LIN {X 0,Y 581.025,Z 523.995,A -85,B 0,C 180,E1 -1875.542,E2 -1875.542} C_VEL
LIN {X 0,Y 580.919,Z 537.737,A -85,B 0,C 180,E1 -1875.999,E2 -1875.999} C_VEL
LIN {X 0,Y 580.786,Z 551.666,A -85,B 0,C 180,E1 -1876.62,E2 -1876.62} C_VEL
LIN {X 0,Y 580.658,Z 564.119,A -85,B 0,C 180,E1 -1877.329,E2 -1877.329} C_VEL
LIN {X 0,Y 580.524,Z 576.656,A -85,B 0,C 180,E1 -1878.213,E2 -1878.213} C_VEL
LIN {X 0,Y 580.44,Z 587.902,A -85,B 0,C 180,E1 -1879.19,E2 -1879.19} C_VEL
LIN {X 0,Y 580.275,Z 597.861,A -85,B 0,C 180,E1 -1880.239,E2 -1880.239} C_VEL
LIN {X 0,Y 580.24,Z 606.18,A -85,B 0,C 180,E1 -1881.293,E2 -1881.293} C_VEL
LIN {X 0,Y 580.165,Z 614.133,A -85,B 0,C 180,E1 -1882.519,E2 -1882.519} C_VEL
LIN {X 0,Y 580.102,Z 620.532,A -85,B 0,C 180,E1 -1883.741,E2 -1883.741} C_VEL
LIN {X 0,Y 580.078,Z 624.965,A -85,B 0,C 180,E1 -1884.788,E2 -1884.788} C_VEL
LIN {X 0,Y 580.102,Z 628.447,A -85,B 0,C 180,E1 -1885.833,E2 -1885.833} C_VEL
LIN {X 0,Y 580.041,Z 631.835,A -85,B 0,C 180,E1 -1887.223,E2 -1887.223} C_VEL
LIN {X 0,Y 580.041,Z 633.834,A -85,B 0,C 180,E1 -1888.612,E2 -1888.612} C_VEL
LIN {X 0,Y 580.036,Z 634.5,A -85,B 0,C 180,E1 -1890.001,E2 -1890.001} C_VEL
LIN {X 0,Y 580.041,Z 633.831,A -85,B 0,C 180,E1 -1891.39,E2 -1891.39} C_VEL
LIN {X 0,Y 580.041,Z 631.829,A -85,B 0,C 180,E1 -1892.779,E2 -1892.779} C_VEL
LIN {X 0,Y 580.102,Z 628.44,A -85,B 0,C 180,E1 -1894.17,E2 -1894.17} C_VEL
LIN {X 0,Y 580.128,Z 623.564,A -85,B 0,C 180,E1 -1895.563,E2 -1895.563} C_VEL
LIN {X 0,Y 580.142,Z 617.048,A -85,B 0,C 180,E1 -1896.959,E2 -1896.959} C_VEL
LIN {X 0,Y 580.192,Z 609.794,A -85,B 0,C 180,E1 -1898.184,E2 -1898.184} C_VEL
LIN {X 0,Y 580.284,Z 600.815,A -85,B 0,C 180,E1 -1899.411,E2 -1899.411} C_VEL
LIN {X 0,Y 580.356,Z 591.382,A -85,B 0,C 180,E1 -1900.467,E2 -1900.467} C_VEL
LIN {X 0,Y 580.479,Z 581.308,A -85,B 0,C 180,E1 -1901.405,E2 -1901.405} C_VEL
LIN {X 0,Y 580.598,Z 569.419,A -85,B 0,C 180,E1 -1902.319,E2 -1902.319} C_VEL
LIN {X 0,Y 580.732,Z 556.628,A -85,B 0,C 180,E1 -1903.116,E2 -1903.116} C_VEL
LIN {X 0,Y 580.873,Z 544.139,A -85,B 0,C 180,E1 -1903.737,E2 -1903.737} C_VEL
LIN {X 0,Y 581.026,Z 531.202,A -85,B 0,C 180,E1 -1904.235,E2 -1904.235} C_VEL
LIN {X 0,Y 581.085,Z 517.151,A -85,B 0,C 180,E1 -1904.632,E2 -1904.632} C_VEL
LIN {X 0,Y 581.166,Z 502.535,A -85,B 0,C 180,E1 -1904.892,E2 -1904.892} C_VEL
LIN {X 0,Y 581.324,Z 376.115,A -85,B 0,C 180,E1 -1906.477,E2 -1906.477} C_VEL
LIN {X 0,Y 580.573,Z 371.811,A -85,B 0,C 180,E1 -1906.574,E2 -1906.574} C_VEL
LIN {X 0,Y 580.774,Z 350.349,A -85,B 0,C 180,E1 -1909.481,E2 -1909.481} C_VEL
LIN {X 0,Y 580.986,Z 329.178,A -85,B 0,C 180,E1 -1912.399,E2 -1912.399} C_VEL
LIN {X 0,Y 580.715,Z 324.205,A -85,B 0,C 180,E1 -1913.107,E2 -1913.107} C_VEL
LIN {X 0,Y 580.269,Z 321.833,A -85,B 0,C 180,E1 -1913.49,E2 -1913.49} C_VEL
LIN {X 0,Y 580.259,Z 321.828,A -85,B 0,C 180,E1 -1916.327,E2 -1916.327} C_VEL
LIN {X 0,Y 580.257,Z 321.832,A -85,B 0,C 180,E1 -1919.302,E2 -1919.302} C_VEL
LIN {X 0,Y 580.287,Z 321.823,A -85,B 0,C 180,E1 -1922.202,E2 -1922.202} C_VEL
LIN {X 0,Y 580.287,Z 321.824,A -85,B 0,C 180,E1 -1924.697,E2 -1924.697} C_VEL
LIN {X 0,Y 580.292,Z 321.83,A -85,B 0,C 180,E1 -1927.27,E2 -1927.27} C_VEL
LIN {X 0,Y 580.298,Z 321.821,A -85,B 0,C 180,E1 -1930.271,E2 -1930.271} C_VEL
LIN {X 0,Y 580.281,Z 321.829,A -85,B 0,C 180,E1 -1932.707,E2 -1932.707} C_VEL
LIN {X 0,Y 580.272,Z 321.824,A -85,B 0,C 180,E1 -1935.61,E2 -1935.61} C_VEL
LIN {X 0,Y 580.285,Z 321.825,A -85,B 0,C 180,E1 -1938.232,E2 -1938.232} C_VEL
LIN {X 0,Y 580.275,Z 321.827,A -85,B 0,C 180,E1 -1940.965,E2 -1940.965} C_VEL
LIN {X 0,Y 580.253,Z 321.826,A -85,B 0,C 180,E1 -1943.595,E2 -1943.595} C_VEL
LIN {X 0,Y 580.316,Z 321.825,A -85,B 0,C 180,E1 -1946.145,E2 -1946.145} C_VEL
LIN {X 0,Y 580.276,Z 321.827,A -85,B 0,C 180,E1 -1948.615,E2 -1948.615} C_VEL
LIN {X 0,Y 580.29,Z 321.823,A -85,B 0,C 180,E1 -1951.024,E2 -1951.024} C_VEL
LIN {X 0,Y 580.251,Z 321.834,A -85,B 0,C 180,E1 -1954.149,E2 -1954.149} C_VEL
LIN {X 0,Y 580.264,Z 321.828,A -85,B 0,C 180,E1 -1956.441,E2 -1956.441} C_VEL
LIN {X 0,Y 580.283,Z 321.886,A -85,B 0,C 180,E1 -1958.415,E2 -1958.415} C_VEL
LIN {X 0,Y 580.722,Z 327.181,A -85,B 0,C 180,E1 -1959.276,E2 -1959.276} C_VEL
LIN {X 0,Y 580.55,Z 345.804,A -85,B 0,C 180,E1 -1962.202,E2 -1962.202} C_VEL
LIN {X 0,Y 580.408,Z 364.473,A -85,B 0,C 180,E1 -1965.089,E2 -1965.089} C_VEL
LIN {X 0,Y 580.367,Z 372.933,A -85,B 0,C 180,E1 -1966.386,E2 -1966.386} C_VEL
LIN {X 0,Y 580.991,Z 377.974,A -85,B 0,C 180,E1 -1966.468,E2 -1966.468} C_VEL
LIN {X 0,Y 580.823,Z 480.346,A -85,B 0,C 180,E1 -1967.753,E2 -1967.753} C_VEL
LIN {X 0,Y 580.758,Z 493.71,A -85,B 0,C 180,E1 -1968.062,E2 -1968.062} C_VEL
LIN {X 0,Y 580.648,Z 505.843,A -85,B 0,C 180,E1 -1968.48,E2 -1968.48} C_VEL
LIN {X 0,Y 580.609,Z 517.266,A -85,B 0,C 180,E1 -1969.01,E2 -1969.01} C_VEL
LIN {X 0,Y 580.451,Z 527.712,A -85,B 0,C 180,E1 -1969.624,E2 -1969.624} C_VEL
LIN {X 0,Y 580.361,Z 538.495,A -85,B 0,C 180,E1 -1970.415,E2 -1970.415} C_VEL
LIN {X 0,Y 580.273,Z 548.158,A -85,B 0,C 180,E1 -1971.292,E2 -1971.292} C_VEL
LIN {X 0,Y 580.222,Z 556.074,A -85,B 0,C 180,E1 -1972.168,E2 -1972.168} C_VEL
LIN {X 0,Y 580.168,Z 563.791,A -85,B 0,C 180,E1 -1973.21,E2 -1973.21} C_VEL
LIN {X 0,Y 580.165,Z 569.111,A -85,B 0,C 180,E1 -1974.09,E2 -1974.09} C_VEL
LIN {X 0,Y 580.053,Z 574.242,A -85,B 0,C 180,E1 -1975.135,E2 -1975.135} C_VEL
LIN {X 0,Y 580.11,Z 578.249,A -85,B 0,C 180,E1 -1976.179,E2 -1976.179} C_VEL
LIN {X 0,Y 580.043,Z 581.184,A -85,B 0,C 180,E1 -1977.222,E2 -1977.222} C_VEL
LIN {X 0,Y 580.038,Z 582.615,A -85,B 0,C 180,E1 -1977.917,E2 -1977.917} C_VEL
LIN {X 0,Y 580.047,Z 583.636,A -85,B 0,C 180,E1 -1978.611,E2 -1978.611} C_VEL
LIN {X 0,Y 580.041,Z 584.263,A -85,B 0,C 180,E1 -1979.306,E2 -1979.306} C_VEL
LIN {X 0,Y 580.038,Z 584.496,A -85,B 0,C 180,E1 -1980,E2 -1980} C_VEL
LIN {X 0,Y 580.04,Z 584.321,A -85,B 0,C 180,E1 -1980.694,E2 -1980.694} C_VEL
LIN {X 0,Y 580.037,Z 582.762,A -85,B 0,C 180,E1 -1982.083,E2 -1982.083} C_VEL
LIN {X 0,Y 580.044,Z 581.392,A -85,B 0,C 180,E1 -1982.778,E2 -1982.778} C_VEL
LIN {X 0,Y 580.11,Z 578.528,A -85,B 0,C 180,E1 -1983.821,E2 -1983.821} C_VEL
LIN {X 0,Y 580.054,Z 574.641,A -85,B 0,C 180,E1 -1984.865,E2 -1984.865} C_VEL
LIN {X 0,Y 580.161,Z 569.585,A -85,B 0,C 180,E1 -1985.91,E2 -1985.91} C_VEL
LIN {X 0,Y 580.158,Z 563.27,A -85,B 0,C 180,E1 -1986.958,E2 -1986.958} C_VEL
LIN {X 0,Y 580.242,Z 555.372,A -85,B 0,C 180,E1 -1988.007,E2 -1988.007} C_VEL
LIN {X 0,Y 580.298,Z 547.29,A -85,B 0,C 180,E1 -1988.883,E2 -1988.883} C_VEL
LIN {X 0,Y 580.364,Z 537.454,A -85,B 0,C 180,E1 -1989.761,E2 -1989.761} C_VEL
LIN {X 0,Y 580.486,Z 526.383,A -85,B 0,C 180,E1 -1990.552,E2 -1990.552} C_VEL
LIN {X 0,Y 580.571,Z 515.562,A -85,B 0,C 180,E1 -1991.168,E2 -1991.168} C_VEL
LIN {X 0,Y 580.675,Z 502.828,A -85,B 0,C 180,E1 -1991.728,E2 -1991.728} C_VEL
LIN {X 0,Y 580.761,Z 489.739,A -85,B 0,C 180,E1 -1992.138,E2 -1992.138} C_VEL
LIN {X 0,Y 580.841,Z 476.222,A -85,B 0,C 180,E1 -1992.402,E2 -1992.402} C_VEL
LIN {X 0,Y 580.932,Z 430.852,A -85,B 0,C 180,E1 -1992.966,E2 -1992.966} C_VEL
LIN {X 0,Y 580.288,Z 425.042,A -85,B 0,C 180,E1 -1993.053,E2 -1993.053} C_VEL
